//Leak Station Not Homed Timeout
GVL_MASTER.stAlarms[2].aEventTimers[0](IN:= (GVL_Master.stStationSruct[2].nState>=200 AND GVL_Master.stStationSruct[2].nState<=900) ,PT:=T#5S);																	
IF GVL_MASTER.stAlarms[2].aEventTimers[0].Q THEN //
	GVL_MASTER.stAlarms[2].aEventFlags[0] := TRUE;
END_IF
//Leak Station Cycle Timeout
GVL_MASTER.stAlarms[2].aEventTimers[1](IN:= (GVL_Master.stStationSruct[2].nState>1000 AND GVL_Master.stStationSruct[2].nState<2000) ,PT:=T#15S);
IF GVL_MASTER.stAlarms[2].aEventTimers[1].Q THEN // 
	GVL_MASTER.stAlarms[2].aEventFlags[1] := TRUE;
END_IF
//Leak Error
GVL_MASTER.stAlarms[2].aEventTimers[2](IN := (NOT PRG_LeakTest.bLeakTesterNoError),PT:=T#100MS);
IF GVL_MASTER.stAlarms[2].aEventTimers[2].Q THEN //
	GVL_MASTER.stAlarms[2].aEventFlags[2] := TRUE;
END_IF
//Consecutive part rejects
IF PRG_LeakTest.nConsParts>2 THEN // 
	GVL_MASTER.stAlarms[2].aEventFlags[3] := TRUE;
END_IF
END_ACTION

METHOD SetEventTexts : BOOL
VAR_INPUT
END_VAR
//Immediate Faults
GVL_MASTER.stAlarms[2].aEventTexts[0] := 'Leak Station Not Homed Timeout';
GVL_MASTER.stAlarms[2].aEventTexts[1] := 'Leak Station Cycle Timeout';
GVL_MASTER.stAlarms[2].aEventTexts[2] := 'Leak Error';
GVL_MASTER.stAlarms[2].aEventTexts[3] := 'More than 2 Consecutive rejects';
GVL_MASTER.stAlarms[2].aEventTexts[4] := '';
GVL_MASTER.stAlarms[2].aEventTexts[5] := '';
GVL_MASTER.stAlarms[2].aEventTexts[6] := '';
GVL_MASTER.stAlarms[2].aEventTexts[7] := '';
GVL_MASTER.stAlarms[2].aEventTexts[8] := '';
GVL_MASTER.stAlarms[2].aEventTexts[9] := ''; 
GVL_MASTER.stAlarms[2].aEventTexts[10] := ''; 
GVL_MASTER.stAlarms[2].aEventTexts[11] := '';
GVL_MASTER.stAlarms[2].aEventTexts[12] := '';
GVL_MASTER.stAlarms[2].aEventTexts[13] := '';
GVL_MASTER.stAlarms[2].aEventTexts[14] := '';
GVL_MASTER.stAlarms[2].aEventTexts[15] := '';
GVL_MASTER.stAlarms[2].aEventTexts[16] := '';
GVL_MASTER.stAlarms[2].aEventTexts[17] := '';
GVL_MASTER.stAlarms[2].aEventTexts[18] := '';
GVL_MASTER.stAlarms[2].aEventTexts[19] := '';
GVL_MASTER.stAlarms[2].aEventTexts[20] := '';
GVL_MASTER.stAlarms[2].aEventTexts[21] := '';
GVL_MASTER.stAlarms[2].aEventTexts[22] := '';
GVL_MASTER.stAlarms[2].aEventTexts[28] := '';
GVL_MASTER.stAlarms[2].aEventTexts[29] := '';
GVL_MASTER.stAlarms[2].aEventTexts[30] := '';

//Cycle Stop Requests

GVL_MASTER.stAlarms[2].aEventTexts[80] := '';
GVL_MASTER.stAlarms[2].aEventTexts[81] := '';
GVL_MASTER.stAlarms[2].aEventTexts[82] := '';

GVL_MASTER.stAlarms[2].aEventTexts[84] := '';
GVL_MASTER.stAlarms[2].aEventTexts[85] := '';
GVL_MASTER.stAlarms[2].aEventTexts[86] := '';
GVL_MASTER.stAlarms[2].aEventTexts[87] := ''; 
GVL_MASTER.stAlarms[2].aEventTexts[88] := '';
GVL_MASTER.stAlarms[2].aEventTexts[89] := '';

//Master Messages

GVL_MASTER.stAlarms[2].aEventTexts[100] := '';
GVL_MASTER.stAlarms[2].aEventTexts[101] := '';
GVL_MASTER.stAlarms[2].aEventTexts[102] := '';
GVL_MASTER.stAlarms[2].aEventTexts[103] := '';
GVL_MASTER.stAlarms[2].aEventTexts[104] := '';
GVL_MASTER.stAlarms[2].aEventTexts[105] := '';
GVL_MASTER.stAlarms[2].aEventTexts[106] := '';
END_METHOD

END_PROGRAM

// ---- POUs/C_LeakTest/PRG_LeakTest.TcPOU
PROGRAM PRG_LeakTest
VAR
	
		TonCaseDelay  		: ARRAY[1..10] OF Tc2_Standard.TON;
		rtrigCaseTriger  	: ARRAY [1..10] OF Tc2_Standard.R_TRIG;
		
		bLeakTesterNoError	: BOOL;
		uCurrentProgramID	: USINT;
		uSetProgramID		: USINT;
		bProgramAccepted	: BOOL;
		bProgramRejected	: BOOL;
		bInstrumentReady	: BOOL;
		bStart				: BOOL;
		bStop				: BOOL;
		bClearErrorIns		: BOOL;
		bTestActiveLiveData	: BOOL;
		nLiveMeasID			: UDINT;
		nLastMeasID			: UDINT;
		bJobPass			: BOOL;
		bJobFailed			: BOOL;
		nConsParts			: INT;






END_VAR
VAR_IN_OUT
	stStationStruct          : ST_StandardStationStruct;
END_VAR

ACT_IOLink();
ACT_TimTrig();

(************** Station in Home Position **************************)
stStationStruct.bStationHomed :=  (stStationStruct.nState = 1000);

(******************************************************************)
stStationStruct.bStationComplete := stStationStruct.nState = 1900;
stStationStruct.bStationHomingRequest := stStationStruct.nState = 200;
stStationStruct.bStationWaitOnRequest := stStationStruct.nState = 1000; 
stStationStruct.bStationInitDone := stStationStruct.nState = 900;
stStationStruct.bStationInProgressInit := stStationStruct.nState >= 200 AND stStationStruct.nState <= 900;
stStationStruct.bStationInProgress :=  stStationStruct.nState > 1000 AND stStationStruct.nState < 1900;
stStationStruct.bStationWaitOnInit := stStationStruct.nState = 100; 
//stStationStruct.bStationAcknowledge := stStationStruct.nState = 200 OR stStationStruct.nState = 1100;
stStationStruct.bStationNotMoving := stStationStruct.nState = 100 OR stStationStruct.nState = 1000 OR stStationStruct.nState = 1900;
(******************************************************************)
(***************** Counter *************)
IF rtrigCaseTriger[1].Q THEN
GVL_PERSIST.stPartsInspection.nLeakPartsGood:= GVL_PERSIST.stPartsInspection.nLeakPartsGood +1;
GVL_PERSIST.stPartsInspection.nLeakTotalPartsGood := GVL_PERSIST.stPartsInspection.nLeakTotalPartsGood+1;
ELSIF GVL_HMI_GLOBAL.bResetLeakGoodParts THEN
GVL_PERSIST.stPartsInspection.nLeakPartsGood:=0;	
END_IF


IF rtrigCaseTriger[2].Q THEN
	GVL_PERSIST.stPartsInspection.nLeakPartsFailed:=GVL_PERSIST.stPartsInspection.nLeakPartsFailed+1;
	GVL_PERSIST.stPartsInspection.nLeakTotalPartsFailed:= GVL_PERSIST.stPartsInspection.nLeakTotalPartsFailed+1;
ELSIF GVL_HMI_GLOBAL.bResetLeakBadParts THEN
	GVL_PERSIST.stPartsInspection.nLeakPartsFailed:=0;
END_IF


bClearErrorIns := GVL_HMI_GLOBAL.bResetButton;

(***************************************)

IF rtrigCaseTriger[3].Q THEN
	stStationStruct.nState := 100;
END_IF

(***************************************)


CASE stStationStruct.nState OF
100: 
bStart							:= FALSE;
IF stStationStruct.bStationInitRequest THEN
	 stStationStruct.nState := 120;
END_IF
120:
bClearErrorIns := TRUE;
IF bClearErrorIns THEN
	stStationStruct.nState := 160;
END_IF
160:
IF tonCaseDelay[2].Q THEN
	bClearErrorIns := FALSE;
	stStationStruct.nState := 180;
END_IF
180: // Check if error 
IF bLeakTesterNoError THEN
	 stStationStruct.nState := 400;
END_IF
400:
IF tonCaseDelay[1].Q THEN
	stStationStruct.nState := 800;
END_IF
800:
IF bInstrumentReady THEN
	stStationStruct.nState := 900;
END_IF
900:
IF stStationStruct.bStationAcknowledge THEN
	stStationStruct.nState := 1000;
END_IF

1000: // Waiting for request 
IF GVL_HMI_GLOBAL.bResetPassAndFail THEN
	GVL_MASTER.stNest.bLeakPass 	:= FALSE;
   GVL_MASTER.stNest.sLeakHMI 	:= "";
   GVL_MASTER.stNest.bLeakReject := FALSE;
END_IF

IF stStationStruct.bStationRequest AND stStationStruct.bNoCycleStopRequest THEN
   stStationStruct.nState := 1100;  
ELSIF (stStationStruct.bStationManualRequestHMI OR GVL_MASTER.bManualModeTrigger) AND stStationStruct.bNoCycleStopRequest THEN
   stStationStruct.nState := 4000; // Manual Mode
ELSIF stStationStruct.bStationAbort THEN
	   stStationStruct.nState := 100;	   
END_IF
1100: // Check Ready
bStart						:= FALSE;
GVL_MASTER.stNest.bLeakPass := FALSE;
GVL_MASTER.stNest.sLeakHMI 	:= "";
IF bInstrumentReady THEN
	stStationStruct.nState := 1140; 
ELSE
	stStationStruct.nState := 100;
END_IF
1140://Check status of intrument
IF bLeakTesterNoError THEN
	stStationStruct.nState := 1200;
END_IF
1200: 
bStart := TRUE;
IF  tonCaseDelay[3].Q THEN
	stStationStruct.nState := 1220;
END_IF
1220:
bStart := FALSE;
IF  NOT bTestActiveLiveData THEN
	stStationStruct.nState := 1280;
END_IF


1280: // JOB PASS / JOB FAIL
IF bJobPass  THEN
	GVL_MASTER.stNest.bLeakPass := TRUE;
	GVL_MASTER.stNest.sLeakHMI 	:= "Pass";
	GVL_MASTER.stNest.bLeakReject := FALSE;
   	stStationStruct.nState := 1900;
ELSIF bJobFailed  THEN
   stStationStruct.nState := 1900;
   GVL_MASTER.stNest.bLeakPass := FALSE;
   GVL_MASTER.stNest.sLeakHMI 	:= "Fail";
   GVL_MASTER.stNest.bLeakReject := TRUE;
END_IF

1900:
IF (tonCaseDelay[4].Q AND NOT stStationStruct.bStationManualRequestHMI) OR stStationStruct.bNoCycleStopRequest THEN
	stStationStruct.nState := 1000;
ELSIF tonCaseDelay[4].Q AND stStationStruct.bStationManualRequestHMI THEN
	stStationStruct.nState := 4000;
ELSIF stStationStruct.bStationAbort AND tonCaseDelay[2].Q THEN
	stStationStruct.nState := 100;

END_IF
//=== Manual Mode ===
4000:
IF NOT stStationStruct.bStationManualRequestHMI AND NOT GVL_MASTER.bManualModeTrigger THEN
	stStationStruct.nState := 1000;
ELSIF stStationStruct.bStationAbort THEN
	   stStationStruct.nState := 100;	
END_IF
IF GVL_HMI_GLOBAL.bStartLeakMan THEN
	
	bStart 						:= TRUE;
ELSIF GVL_HMI_GLOBAL.bStopLeakMan THEN
	
	bStop						:= TRUE;

ELSE 
	bStart						:= FALSE;
	bStop						:= FALSE;
END_IF
ACT_ChangeJOB();

9000:

bClearErrorIns 					:= FALSE;
bStart							:= FALSE;
GVL_MASTER.stNest.bLeakPass 	:= FALSE;


stStationStruct.nState := 9100;	
9100:
IF tonCaseDelay[5].Q THEN
	stStationStruct.nState := 9200;
END_IF
9200:
bClearErrorIns := TRUE;
IF tonCaseDelay[6].Q THEN
	stStationStruct.nState := 9300;
END_IF
9300: 
IF bLeakTesterNoError THEN
   stStationStruct.nState := 1000;
END_IF

	
END_CASE

IF NOT bLeakTesterNoError AND NOT stStationStruct.nState >= 9000 THEN
stStationStruct.nState := 9000;
END_IF

ACTION ACT_ChangeJob:
	
GVL_IO.dw_B07_i28General_I_O.bSetProgram[0] := GVL_HMI_GLOBAL.uNewLeakProgID.0;
GVL_IO.dw_B07_i28General_I_O.bSetProgram[1] := GVL_HMI_GLOBAL.uNewLeakProgID.1;
GVL_IO.dw_B07_i28General_I_O.bSetProgram[2] := GVL_HMI_GLOBAL.uNewLeakProgID.2;
GVL_IO.dw_B07_i28General_I_O.bSetProgram[3] := GVL_HMI_GLOBAL.uNewLeakProgID.3;
GVL_IO.dw_B07_i28General_I_O.bSetProgram[4] := GVL_HMI_GLOBAL.uNewLeakProgID.4;
GVL_IO.dw_B07_i28General_I_O.bSetProgram[5] := GVL_HMI_GLOBAL.uNewLeakProgID.5;
GVL_IO.dw_B07_i28General_I_O.bSetProgram[6] := GVL_HMI_GLOBAL.uNewLeakProgID.6;
GVL_IO.dw_B07_i28General_I_O.bSetProgram[7] := GVL_HMI_GLOBAL.uNewLeakProgID.7;


IF GVL_HMI_GLOBAL.bSetLeakProgramID THEN 
	
		uSetProgramID := GVL_HMI_GLOBAL.uNewLeakProgID;
END_IF
END_ACTION

ACTION ACT_IOLINK:


bLeakTesterNoError				:= NOT GVL_IO.dw_B07_i28General_I_O.bMalfunction;
uCurrentProgramID				:= GVL_IO.dw_B07_i28General_I_O.nCurrentProgramNumber;
bProgramAccepted				:= GVL_IO.dw_B07_i28General_I_O.bProgramAccept;
bInstrumentReady				:= GVL_IO.dw_B07_i28General_I_O.bInstrumentReady;
bProgramRejected				:= GVL_IO.dw_B07_i28General_I_O.bProgramReject;
bTestActiveLiveData				:= GVL_IO.dw_B07_i28General_I_O.bTestActiveLiveData;
nLiveMeasID						:= GVL_IO.dw_B07_i28LiveMeasurement.inUniqueID;
nLastMeasID						:= GVL_IO.dw_B07_i28LastResult.inUniqueID;
bJobPass						:= GVL_IO.dw_B07_i28General_I_O.bProgramAccept;
bJobFailed						:= GVL_IO.dw_B07_i28General_I_O.bProgramReject;



GVL_IO.dw_B07_i28General_I_O.bStart 			:= bStart;
GVL_IO.dw_B07_i28General_I_O.bStop				:= bStop;
GVL_IO.dw_B07_i28General_I_O.bChangeProgram := GVL_HMI_GLOBAL.bSetLeakProgramID;
GVL_IO.dw_B07_i28General_I_O.bReset := bClearErrorIns OR GVL_HMI_GLOBAL.bResetLeakMan;
END_ACTION

ACTION ACT_TimTrig:


tonCaseDelay[1](IN:= (stStationStruct.nState=400),PT:=T#50MS);
tonCaseDelay[2](IN:= (stStationStruct.nState=160),PT:=T#50MS);
tonCaseDelay[3](IN:= (stStationStruct.nState=1200),PT:=T#10S);
tonCaseDelay[4](IN:= (stStationStruct.nState=1900),PT:=T#1S);
tonCaseDelay[5](IN:= (stStationStruct.nState=9100),PT:=T#200MS);
tonCaseDelay[6](IN:= (stStationStruct.nState=9200),PT:=T#250MS);
tonCaseDelay[7](IN:= ,PT:=T#500MS);



rtrigCaseTriger[1](clk:= (stStationStruct.nState=1900) AND bJobPass);
rtrigCaseTriger[2](clk:= (stStationStruct.nState=1900) AND bJobFailed);
rtrigCaseTriger[3](clk:= stStationStruct.bStationAbort);
END_ACTION

END_PROGRAM

// ---- POUs/D_VisionTest/PRG_Fault_VisionTest.TcPOU
PROGRAM PRG_Fault_VisionTest
VAR
	
			i				: INT;
			
END_VAR
VAR_IN_OUT

  aAlarms  : ARRAY[0..3] OF ST_Events;
END_VAR

ACT_FaultTrig();

(************************************** Faults reset **********************************************)
IF   GVL_HMI_GLOBAL.bResetButton THEN 
	FOR i := 0 TO 127 DO
		GVL_MASTER.stAlarms[3].aEventFlags[i] := FALSE;
	END_FOR
END_IF
//===============================================================
//Initialize event texts on first scan
IF NOT GVL_MASTER.stAlarms[3].bEventTextsSet THEN
	SetEventTexts();
	GVL_MASTER.stAlarms[3].bEventTextsSet := TRUE;
END_IF


(***************************************************************************************************)
//Immediate fault
GVL_MASTER.stAlarms[3].bImmediateFault := FALSE;
FOR i := 0 TO 32DO
	GVL_MASTER.stAlarms[3].bImmediateFault := GVL_MASTER.stAlarms[3].bImmediateFault OR GVL_MASTER.stAlarms[3].aEventFlags[i];
END_FOR

//Cycle stop fault
GVL_MASTER.stAlarms[3].bCycleStopFault := FALSE;
FOR i := 33 TO 79 DO
	GVL_MASTER.stAlarms[3].bCycleStopFault := GVL_MASTER.stAlarms[3].bCycleStopFault OR GVL_MASTER.stAlarms[3].aEventFlags[i];
END_FOR
//Cycle stop Request
GVL_MASTER.stAlarms[3].bCycleStopRequest := FALSE;
FOR i := 80 TO 99 DO
	GVL_MASTER.stAlarms[3].bCycleStopRequest := GVL_MASTER.stAlarms[3].bCycleStopRequest OR GVL_MASTER.stAlarms[3].aEventFlags[i];
END_FOR

ACTION ACT_FaultTrig:
(**************************************************************************************************)
(**************************** Master Immediate Fault Stop *****************************************)
(**************************************************************************************************)
(* Copy Safety Immediate Stop Faults to Master Immediate Stop Faults *)
(* *)

//Camera Station Not Homed Timeout
GVL_MASTER.stAlarms[3].aEventTimers[0](IN:= (GVL_Master.stStationSruct[3].nState>=200 AND GVL_Master.stStationSruct[3].nState<=900) ,PT:=T#5S);																	
IF GVL_MASTER.stAlarms[3].aEventTimers[0].Q THEN //
	GVL_MASTER.stAlarms[3].aEventFlags[0] := TRUE;
END_IF
//Camera Station Cycle Timeout
GVL_MASTER.stAlarms[3].aEventTimers[1](IN:= (GVL_Master.stStationSruct[3].nState>=1100 AND GVL_Master.stStationSruct[3].nState<1900) ,PT:=T#5S);
IF GVL_MASTER.stAlarms[3].aEventTimers[1].Q THEN // 
	GVL_MASTER.stAlarms[3].aEventFlags[1] := TRUE;
END_IF
//Camera Error
GVL_MASTER.stAlarms[3].aEventTimers[2](IN := (NOT PRG_VisionTest.bCamerraNoError),PT:=T#100MS);
IF GVL_MASTER.stAlarms[3].aEventTimers[2].Q THEN //
	GVL_MASTER.stAlarms[3].aEventFlags[2] := TRUE;
END_IF
//Consecutive part rejects
(*IF PRG_VisionTest.nConsParts>2 THEN // 
	GVL_MASTER.stAlarms[3].aEventFlags[3] := TRUE;
END_IF*)

//Adquisition error
IF GVL_IO.dw_B06_IS2802M.aqsAcquisitionError  THEN
	GVL_MASTER.stAlarms[3].aEventFlags[100] := TRUE;
ELSIF NOT GVL_IO.dw_B06_IS2802M.aqsAcquisitionError THEN
   	GVL_MASTER.stAlarms[3].aEventFlags[100] := FALSE;
END_IF
END_ACTION

METHOD PRIVATE SetEventTexts : BOOL
VAR_INPUT
END_VAR
//Immediate Faults
GVL_MASTER.stAlarms[3].aEventTexts[0] := 'Camera Station Not Homed Timeout';
GVL_MASTER.stAlarms[3].aEventTexts[1] := 'Camera Station Cycle Timeout';
GVL_MASTER.stAlarms[3].aEventTexts[2] := 'Camera Error';
//GVL_MASTER.stAlarms[3].aEventTexts[3] := 'More than 2 Consecutive rejects';
GVL_MASTER.stAlarms[3].aEventTexts[4] := '';
GVL_MASTER.stAlarms[3].aEventTexts[5] := '';
GVL_MASTER.stAlarms[3].aEventTexts[6] := '';
GVL_MASTER.stAlarms[3].aEventTexts[7] := '';
GVL_MASTER.stAlarms[3].aEventTexts[8] := '';
GVL_MASTER.stAlarms[3].aEventTexts[9] := ''; 
GVL_MASTER.stAlarms[3].aEventTexts[10] := ''; 
GVL_MASTER.stAlarms[3].aEventTexts[11] := '';
GVL_MASTER.stAlarms[3].aEventTexts[12] := '';
GVL_MASTER.stAlarms[3].aEventTexts[13] := '';
GVL_MASTER.stAlarms[3].aEventTexts[14] := '';
GVL_MASTER.stAlarms[3].aEventTexts[15] := '';
GVL_MASTER.stAlarms[3].aEventTexts[16] := '';
GVL_MASTER.stAlarms[3].aEventTexts[17] := '';
GVL_MASTER.stAlarms[3].aEventTexts[18] := '';
GVL_MASTER.stAlarms[3].aEventTexts[19] := '';
GVL_MASTER.stAlarms[3].aEventTexts[20] := '';
GVL_MASTER.stAlarms[3].aEventTexts[21] := '';
GVL_MASTER.stAlarms[3].aEventTexts[22] := '';
GVL_MASTER.stAlarms[3].aEventTexts[28] := '';
GVL_MASTER.stAlarms[3].aEventTexts[29] := '';
GVL_MASTER.stAlarms[3].aEventTexts[30] := '';

//Cycle Stop Requests

GVL_MASTER.stAlarms[3].aEventTexts[80] := '';
GVL_MASTER.stAlarms[3].aEventTexts[81] := '';
GVL_MASTER.stAlarms[3].aEventTexts[82] := '';

GVL_MASTER.stAlarms[3].aEventTexts[84] := '';
GVL_MASTER.stAlarms[3].aEventTexts[85] := '';
GVL_MASTER.stAlarms[3].aEventTexts[86] := '';
GVL_MASTER.stAlarms[3].aEventTexts[87] := ''; 
GVL_MASTER.stAlarms[3].aEventTexts[88] := '';
GVL_MASTER.stAlarms[3].aEventTexts[89] := '';

//Master Messages

GVL_MASTER.stAlarms[3].aEventTexts[100] := 'Acquisition Error';
GVL_MASTER.stAlarms[3].aEventTexts[101] := '';
GVL_MASTER.stAlarms[3].aEventTexts[102] := '';
GVL_MASTER.stAlarms[3].aEventTexts[103] := '';
GVL_MASTER.stAlarms[3].aEventTexts[104] := '';
GVL_MASTER.stAlarms[3].aEventTexts[105] := '';
GVL_MASTER.stAlarms[3].aEventTexts[106] := '';
END_METHOD

END_PROGRAM

// ---- POUs/D_VisionTest/PRG_VisionTest.TcPOU
PROGRAM PRG_VisionTest
VAR

	biClamp				: BOOL;

	rTrigJobChangeReq	: R_TRIG;
	rTrigProdJob		: R_TRIG;
	rTrigCalibJob		: R_TRIG;

	bCommandExecuting	: BOOL;
	bCommandFailed		: BOOL;
	bCommandCompleted 	: BOOL;
	bCommandExecute		: BOOL;
	nCommandID			: UINT;
	bCamerraNoError     : BOOL;
	bCameraBufOverR     : BOOL;
	bInspectionCompleted: RS;
	bResultValid        : BOOL;
	bJobPass            : BOOL;
	bAqusError          : BOOL;
	bExposComplete      : BOOL;
	bAqusTriggerReady   : BOOL;
	bOnline             : BOOL;
	bOffline            : BOOL;
	bEnableTrigger      : BOOL;
	bTriggerCam         : BOOL;
	bComplete           : BOOL;
	bClearCamError      : BOOL;
	bAcnwResult         : BOOL;
	nCammeraErrorID     : UINT;	
	nAqusID             : UINT;
	nCurrentJobID       : UINT;	
	nRempAqusID         : UINT;
	nCameraJob          : UINT := 1;
	nAqusID_Temp        : UINT := 0;
	bManPass            : BOOL;
	bManFail            : BOOL;
	bManEnablTrig       : BOOL;
	bManTrigCam         : BOOL;
	bManAknwResult      : BOOL;
	bManComplResl       : BOOL;	
	
	nCoutAqErr			: INT;

		
	TonCaseDelay  		: ARRAY[1..10] OF Tc2_Standard.TON;
	rtrigCaseTriger  	: ARRAY [1..10] OF Tc2_Standard.R_TRIG;
	adbCaseFlag      	: ARRAY [1..10] OF BOOL;
	eCamJobState		: E_CameraJobChange;

	nConsParts			: INT;
END_VAR

VAR_IN_OUT
	stStationStruct     : ST_StandardStationStruct;
END_VAR

ACT_IOLink();
ACT_ChangeJob();
ACT_TimTrig();

(************** Station in Home Position **************************)
stStationStruct.bStationHomed :=  (stStationStruct.nState = 1000);

(******************************************************************)
stStationStruct.bStationComplete := stStationStruct.nState = 1900;
stStationStruct.bStationHomingRequest := stStationStruct.nState = 200;
stStationStruct.bStationWaitOnRequest := stStationStruct.nState = 1000; 
stStationStruct.bStationInitDone := stStationStruct.nState = 900;
stStationStruct.bStationInProgressInit := stStationStruct.nState >= 200 AND stStationStruct.nState <= 900;
stStationStruct.bStationInProgress :=  stStationStruct.nState > 1000 AND stStationStruct.nState < 1900;
stStationStruct.bStationWaitOnInit := stStationStruct.nState = 100; 
//stStationStruct.bStationAcknowledge := stStationStruct.nState = 200 OR stStationStruct.nState = 1100;
stStationStruct.bStationNotMoving := stStationStruct.nState = 100 OR stStationStruct.nState = 1000 OR stStationStruct.nState = 1900;
(******************************************************************)
(***************** Counter *************)
IF rtrigCaseTriger[3].Q THEN
GVL_PERSIST.stPartsInspection.nVisionPartsGood:= GVL_PERSIST.stPartsInspection.nVisionPartsGood +1;
GVL_PERSIST.stPartsInspection.nVisionTotalPartsGood := GVL_PERSIST.stPartsInspection.nVisionTotalPartsGood+1;
ELSIF GVL_HMI_GLOBAL.bResetVisionGoodParts THEN
GVL_PERSIST.stPartsInspection.nVisionPartsGood:=0;	
END_IF


IF rtrigCaseTriger[4].Q THEN
	GVL_PERSIST.stPartsInspection.nVisionPartsFailed:=GVL_PERSIST.stPartsInspection.nVisionPartsFailed+1;
	GVL_PERSIST.stPartsInspection.nVisionTotalPartsFailed:= GVL_PERSIST.stPartsInspection.nVisionTotalPartsFailed+1;
ELSIF GVL_HMI_GLOBAL.bResetVisionBadParts THEN
	GVL_PERSIST.stPartsInspection.nVisionPartsFailed:=0;
END_IF

IF rtrigCaseTriger[4].Q THEN
	nConsParts:= nConsParts+1;
ELSIF rtrigCaseTriger[3].Q OR GVL_HMI_GLOBAL.bResetButton THEN
    nConsParts:=0;	
END_IF

bClearCamError := GVL_HMI_GLOBAL.bResetButton;

(***************************************)

IF rtrigCaseTriger[5].Q THEN
	stStationStruct.nState := 100;
END_IF

(***************************************)


CASE stStationStruct.nState OF
100: 
IF stStationStruct.bStationInitRequest THEN
	 stStationStruct.nState := 140;
END_IF
140:
bClearCamError := TRUE;
IF bClearCamError THEN
	stStationStruct.nState := 160;
END_IF
160:
IF tonCaseDelay[8].Q THEN
	bClearCamError := FALSE;
	stStationStruct.nState := 200;
END_IF
200: // Check if error 
IF bCamerraNoError THEN
	 stStationStruct.nState := 400;
END_IF
300: // Check ID job
IF nCurrentJobID = nCameraJob THEN
	stStationStruct.nState := 400;
END_IF
400:
IF tonCaseDelay[1].Q THEN
	stStationStruct.nState := 900;
END_IF
900:
IF stStationStruct.bStationAcknowledge THEN
	stStationStruct.nState := 1000;
END_IF
1000: // Waiting for request 
adbCaseFlag[1] := FALSE;
adbCaseFlag[2] := FALSE;
bEnableTrigger := FALSE;
bTriggerCam    := FALSE;

bAcnwResult := FALSE;
bComplete:= FALSE;
IF GVL_HMI_GLOBAL.bResetPassAndFail THEN
	GVL_MASTER.stNest.bVisionPass := FALSE;
	GVL_MASTER.stNest.sVisionHMI := "";
	GVL_MASTER.stNest.bVisionReject := FALSE;
END_IF
IF stStationStruct.bStationRequest AND stStationStruct.bNoCycleStopRequest THEN
   stStationStruct.nState := 1100;  
ELSIF (stStationStruct.bStationManualRequestHMI OR GVL_MASTER.bManualModeTrigger) AND stStationStruct.bNoCycleStopRequest THEN
   stStationStruct.nState := 4000; // Manual Mode
ELSIF stStationStruct.bStationAbort THEN
	   stStationStruct.nState := 100;	   
END_IF
1100:// Check Buffer
IF NOT bCameraBufOverR THEN
	stStationStruct.nState := 1160;
ELSIF bCameraBufOverR THEN
	stStationStruct.nState := 1120;  
END_IF
1120: 
bOffline := TRUE;
IF NOT bOnline THEN
	bClearCamError := TRUE;
	stStationStruct.nState := 1130; 
END_IF
1130:
IF bClearCamError THEN
	bClearCamError := FALSE;
	stStationStruct.nState := 1140;
END_IF
1140:
IF NOT bClearCamError THEN
       bOffline := FALSE;
       stStationStruct.nState := 1160; 
END_IF
1160: // Check ofline/online
IF bOnline THEN
	stStationStruct.nState := 1200; 
ELSE
	adbCaseFlag[1] := TRUE;
    stStationStruct.nState := 1200; 
END_IF
1180://Check status if Cam
IF nCammeraErrorID =0 THEN
	stStationStruct.nState := 1200;
ELSE
    adbCaseFlag[2] := TRUE;	
	stStationStruct.nState := 2000;
END_IF
1200://Enable Trigger
bEnableTrigger := TRUE;
IF bAqusTriggerReady THEN
	stStationStruct.nState := 1220;
END_IF
1220: 
bTriggerCam := TRUE;
IF  bExposComplete THEN
	stStationStruct.nState := 1240;
END_IF
1240:
IF bResultValid THEN
	bEnableTrigger := FALSE;
	bTriggerCam := FALSE;
	stStationStruct.nState := 1260;
END_IF
1260:// Check Aqusition
IF nAqusID<> nAqusID_Temp AND bInspectionCompleted.Q1 THEN
	stStationStruct.nState := 1270;
END_IF
1270:
IF tonCaseDelay[9].Q THEN
	stStationStruct.nState := 1280;
END_IF

1280: // JOB PASS / JOB FAIL
IF bJobPass  THEN
//   nPartStatus := 1;
	GVL_MASTER.stNest.bVisionPass 	:= TRUE;
	GVL_MASTER.stNest.sVisionHMI 	:= "Pass";
   stStationStruct.nState := 1300;
ELSIF NOT bJobPass  THEN
	//Added checks here not initial for bNestFail or bNestPartReject	
//   nPartStatus := 0;
   GVL_MASTER.stNest.bVisionReject := TRUE;
   GVL_MASTER.stNest.sVisionHMI 	:= "Fail";
   stStationStruct.nState := 1282;
END_IF
1282:
bAcnwResult := TRUE;
IF NOT bResultValid THEN
	stStationStruct.nState := 1284;
END_IF
1284:
bAcnwResult := FALSE;
IF NOT bAcnwResult AND NOT bResultValid THEN
	nAqusID_Temp:= nAqusID;
	stStationStruct.nState := 1286;
END_IF
1286:
bComplete:= TRUE;
IF NOT bExposComplete THEN
	stStationStruct.nState := 1288;
END_IF
1288:
bComplete:= FALSE;
IF NOT bComplete AND NOT bExposComplete THEN
	stStationStruct.nState := 1290;
END_IF	
1290:
adbCaseFlag[1] := FALSE;
adbCaseFlag[2] := FALSE;
bEnableTrigger := FALSE;
bTriggerCam    := FALSE;
bAcnwResult := FALSE;
bComplete:= FALSE;
stStationStruct.nState := 1292;
1292:
bEnableTrigger := TRUE;
IF bEnableTrigger AND tonCaseDelay[7].Q THEN
	stStationStruct.nState := 1294;
END_IF
1294:
bTriggerCam := TRUE;
IF  bExposComplete THEN
	stStationStruct.nState := 1296;
END_IF
1296:
IF bResultValid THEN
	bEnableTrigger := FALSE;
    bTriggerCam := FALSE;
    stStationStruct.nState := 1298;
END_IF
1298:
IF bJobPass  THEN
//   nPartStatus := 1;
   stStationStruct.nState := 1300;
ELSIF NOT  bJobPass THEN
//   nPartStatus := 0;
   stStationStruct.nState := 1300;
END_IF

1300:
bAcnwResult := TRUE;
IF NOT bResultValid THEN
	stStationStruct.nState := 1320;
END_IF
1320:
bAcnwResult := FALSE;
IF NOT bAcnwResult AND NOT bResultValid THEN
	nAqusID_Temp:= nAqusID;
	stStationStruct.nState := 1340;
END_IF
1340:
bComplete:= TRUE;
IF NOT bExposComplete THEN
	stStationStruct.nState := 1360;
END_IF
1360:
bComplete:= FALSE;
IF NOT bComplete AND NOT bExposComplete THEN
	stStationStruct.nState := 1900;
END_IF	
1900:
adbCaseFlag[1] := FALSE;
adbCaseFlag[2] := FALSE;
bEnableTrigger := FALSE;
bTriggerCam    := FALSE;
bAcnwResult := FALSE;
bComplete:= FALSE;
IF tonCaseDelay[2].Q AND rtrigCaseTriger[7].Q THEN
	stStationStruct.nState := 1000;
ELSIF NOT stStationStruct.bNoCycleStopRequest AND tonCaseDelay[2].Q THEN
	stStationStruct.nState := 1000;
END_IF
//=== Manual Mode ===
4000:
IF NOT stStationStruct.bStationManualRequestHMI  AND NOT GVL_MASTER.bManualModeTrigger THEN
	stStationStruct.nState := 1000;
END_IF
IF GVL_HMI_GLOBAL.bEnableTrigerMan THEN
	bManEnablTrig := TRUE;
	bManPass:= FALSE;
	bManFail:= FALSE;
	stStationStruct.nState := 4100;
ELSIF stStationStruct.bStationAbort THEN
	   stStationStruct.nState := 100;		
END_IF
4100:
	bManPass:= FALSE;
	bManFail:= FALSE;
IF NOT stStationStruct.bStationManualRequestHMI THEN
	bManEnablTrig := FALSE;
	stStationStruct.nState := 1000;
ELSIF stStationStruct.bStationAbort THEN
	   bManEnablTrig := FALSE;
	   stStationStruct.nState := 100;		
ELSIF GVL_HMI_GLOBAL.bTrigerCamMan THEN
	GVL_HMI_GLOBAL.bEnableTrigerMan:= FALSE;
	bManTrigCam := TRUE;
	stStationStruct.nState := 4200;
END_IF
4200:
GVL_HMI_GLOBAL.bTrigerCamMan := FALSE;
IF  bExposComplete THEN
	stStationStruct.nState := 4300;
END_IF
4300:
IF bResultValid THEN
	bManEnablTrig := FALSE;
    bManTrigCam := FALSE;
    stStationStruct.nState := 4400;
END_IF
4400:
IF bJobPass THEN
	bManPass := TRUE;
	bManFail := FALSE;
//	nPartStatus := 1;
	stStationStruct.nState := 4500;
ELSIF NOT bJobPass  THEN
	bManPass := FALSE;
	bManFail := TRUE;
//	nPartStatus := 0;
	stStationStruct.nState := 4500;
END_IF
4500:
bManAknwResult := TRUE;
IF NOT bResultValid THEN
	stStationStruct.nState := 4600;
END_IF
4600:
bManAknwResult := FALSE;
bManComplResl := TRUE;
IF NOT bExposComplete THEN
	stStationStruct.nState := 4700;
END_IF
4700:
bManAknwResult := FALSE;
bManComplResl  := FALSE;
bManEnablTrig  := FALSE;
bManTrigCam    := FALSE;
IF NOT stStationStruct.bStationManualRequestHMI THEN
stStationStruct.nState := 4000;
ELSE
stStationStruct.nState := 1000;	
END_IF
9000:

bManAknwResult := FALSE;
bManComplResl  := FALSE;
bManEnablTrig  := FALSE;
bManTrigCam    := FALSE;	
bOffline       := FALSE;
bEnableTrigger := FALSE;
bTriggerCam    := FALSE;
bComplete      := FALSE;
bClearCamError := FALSE;
bAcnwResult    := FALSE;
stStationStruct.nState := 9100;	
9100:
IF tonCaseDelay[5].Q THEN
	stStationStruct.nState := 9200;
END_IF
9200:
bClearCamError := TRUE;
IF tonCaseDelay[6].Q THEN
	stStationStruct.nState := 9300;
END_IF
9300: 
IF nCoutAqErr >3 THEN
   stStationStruct.nState := 1000;
ELSIF nCoutAqErr <=3 THEN
   stStationStruct.nState := 1100;
END_IF

	
END_CASE

IF bAqusError AND NOT stStationStruct.nState >= 9000 THEN
stStationStruct.nState := 9000;
END_IF


IF rtrigCaseTriger[6].Q THEN
   nCoutAqErr := nCoutAqErr +1;
ELSIF  stStationStruct.nState = 1000 THEN
    nCoutAqErr := 0;
END_IF

ACTION ACT_ChangeJob:
rTrigProdJob(CLK := GVL_HMI_GLOBAL.bLoadProductionJob);
rTrigCalibJob(CLK := GVL_HMI_GLOBAL.bLoadCalibrationJob);

IF rTrigProdJob.Q THEN
	eCamJobState := E_CameraJobChange.LOAD_PROD_JOB;
END_IF

IF rTrigCalibJob.Q THEN
	eCamJobState := E_CameraJobChange.LOAD_CALB_JOB;
END_IF

CASE eCamJobState OF
	
E_CameraJobChange.WAITING_FOR_REQUEST:
//Do nothing

E_CameraJobChange.LOAD_PROD_JOB:
	(*Load Production Job*)
	nCommandID := 1;
	eCamJobState := E_CameraJobChange.GO_OFFLINE;

E_CameraJobChange.LOAD_CALB_JOB:
	(*Load Calibration Job*)
	nCommandID := 101;
	eCamJobState := E_CameraJobChange.GO_OFFLINE;

E_CameraJobChange.GO_OFFLINE:
	bOffline := TRUE;
	eCamJobState := E_CameraJobChange.EXECUTE_COMMAND;

E_CameraJobChange.EXECUTE_COMMAND:
	bCommandExecute := TRUE;
	eCamJobState := E_CameraJobChange.RESET_FLAG;
	
E_CameraJobChange.RESET_FLAG:
IF bCommandCompleted THEN
	bCommandExecute := FALSE;
	bOffline := FALSE;
	GVL_HMI_GLOBAL.bLoadProductionJob := FALSE;
	GVL_HMI_GLOBAL.bLoadCalibrationJob := FALSE;
	eCamJobState := E_CameraJobChange.WAITING_FOR_REQUEST;
END_IF
END_CASE
END_ACTION

ACTION ACT_IOLink:

bCamerraNoError      := NOT GVL_IO.dw_B06_IS2802M.isError;//==
nCammeraErrorID      := GVL_IO.dw_B06_IS2802M.isErrorID;//--nchamera UI
bCameraBufOverR      := GVL_IO.dw_B06_IS2802M.isResultsBufferOverrun;
bInspectionCompleted(SET := GVL_IO.dw_B06_IS2802M.isInspectionCompleted, RESET1 := stStationStruct.nState > 1260);
bResultValid         := GVL_IO.dw_B06_IS2802M.isResultsValid;
bJobPass             := GVL_IO.dw_B06_IS2802M.isJobPassed;
bAqusError           := GVL_IO.dw_B06_IS2802M.aqsAcquisitionError;
bExposComplete       := GVL_IO.dw_B06_IS2802M.aqsExposureComplete;
bAqusTriggerReady    := GVL_IO.dw_B06_IS2802M.aqsTriggerReady;
bOnline              := GVL_IO.dw_B06_IS2802M.aqsOnline;
nAqusID              := GVL_IO.dw_B06_IS2802M.aqsAcquisitionID;
nCurrentJobID        := GVL_IO.dw_B06_IS2802M.ccoCurrentJobID;
bCommandExecuting	 := GVL_IO.dw_B06_IS2802M.isCommandExecuting;
bCommandFailed		 := GVL_IO.dw_B06_IS2802M.isCommandFailed;
bCommandCompleted    := GVL_IO.dw_B06_IS2802M.isCommandCompleted;
GVL_IO.dw_B06_IS2802M.aqcSetOffline                  := bOffline;
GVL_IO.dw_B06_IS2802M.aqcTriggerEnable               := bEnableTrigger OR bManEnablTrig;
GVL_IO.dw_B06_IS2802M.aqcTrigger                     := bTriggerCam OR bManTrigCam;
GVL_IO.dw_B06_IS2802M.aqcClearExposureComplete       := bComplete OR bManComplResl;
GVL_IO.dw_B06_IS2802M.icClearError                   := bClearCamError OR GVL_HMI_GLOBAL.bResetCamMan ;//--
GVL_IO.dw_B06_IS2802M.icInspectionResultsAcknowledge := bAcnwResult OR bManAknwResult ;
GVL_IO.dw_B06_IS2802M.cciCommandID					 := nCommandID;
GVL_IO.dw_B06_IS2802M.icExecuteCommand				 := bCommandExecute;

biClamp					:= GVL_IO.dw_T02_EL1809.iCalmpClosed;

IF tonCaseDelay[4].Q THEN
	GVL_HMI_GLOBAL.bResetCamMan:= FALSE;
END_IF

IF NOT bExposComplete THEN
   bComplete:= FALSE;
END_IF
IF bExposComplete THEN
	bTriggerCam := FALSE;
END_IF
IF NOT bResultValid THEN
	bAcnwResult := FALSE;
END_IF

IF NOT GVL_Master.stMachineStatus.bManualMode THEN
   GVL_HMI_GLOBAL.sInfoCamMan:= 'Machine not in Manual Mode';
ELSIF GVL_Master.stMachineStatus.bManualMode AND stStationStruct.nState>4100 THEN
   GVL_HMI_GLOBAL.sInfoCamMan:= 'Camera in Process';
ELSIF  GVL_Master.stMachineStatus.bManualMode AND stStationStruct.nState=4000 THEN
   GVL_HMI_GLOBAL.sInfoCamMan:= 'Waiting for Enable'; 
ELSIF  GVL_Master.stMachineStatus.bManualMode AND stStationStruct.nState=4100 THEN
   GVL_HMI_GLOBAL.sInfoCamMan:= 'Waiting for Trigger';		   
END_IF
END_ACTION

ACTION ACT_TimTrig:
tonCaseDelay[1](IN:= (stStationStruct.nState=400),PT:=T#50MS);
tonCaseDelay[2](IN:= (stStationStruct.nState=1900),PT:=T#100MS);
tonCaseDelay[3](IN:= (stStationStruct.nState=1),PT:=T#100MS);
tonCaseDelay[4](IN:= GVL_HMI_GLOBAL.bResetCamMan,PT:=T#100MS);
tonCaseDelay[5](IN:= (stStationStruct.nState=9100),PT:=T#250MS);
tonCaseDelay[6](IN:= (stStationStruct.nState=9200),PT:=T#250MS);
tonCaseDelay[7](IN:= (stStationStruct.nState=1292),PT:=T#50MS);
tonCaseDelay[8](IN:= (stStationStruct.nState=160),PT:=T#250MS);
tonCaseDelay[9](IN:=stStationStruct.nState=1270 ,PT:=T#1S);
tonCaseDelay[10](IN:= ,PT:=T#250MS);

rtrigCaseTriger[1](clk:= stStationStruct.nState>1100);
rtrigCaseTriger[2](clk:= adbCaseFlag[1]);
rtrigCaseTriger[3](clk:= (stStationStruct.nState=1900) AND bJobPass );
rtrigCaseTriger[4](clk:= (stStationStruct.nState=1900) AND NOT bJobPass );
rtrigCaseTriger[5](clk:= stStationStruct.bStationAbort);
rtrigCaseTriger[6](clk:= (stStationStruct.nState=1240) AND  bAqusError );
rtrigCaseTriger[7](clk:= biClamp);
rtrigCaseTriger[8](clk:= );
rtrigCaseTriger[9](clk:= );
rtrigCaseTriger[10](clk:= );
END_ACTION

END_PROGRAM

// ---- POUs/A_Master/PRG_MachineStatus.TcPOU
PROGRAM PRG_MachineStatus
VAR

	tonPowerUp						: TON;
	tonSystemInitialising			: TON;
	tonSystemInitialisingTimeout	: TON;
	
	bMemoSystemReadyToStart			:BOOL; //flag set only once to establissh if system was in ready to start state after powerUP
	
// =========== Manual =============	

	rtrigManualModeOFF              :ARRAY[1..4] OF R_TRIG;
	rtrigManualMode                 :R_TRIG;	
		// =========== Master Time =============
		//Variables
	bReadyToRead				:BOOL;
	bFirstScan					:BOOL := TRUE;
	bUpdateSysTime				:BOOL; //Output of pulse generator
	tSysTimeUpdatePeriod		:TIME := T#5S;
	stTimeStamp					:TIMESTRUCT;
	stNullTimeStamp				:TIMESTRUCT;
	sRawDateTime				:STRING;

	

	
	
	sDateTime					:STRING;
	sDateTimeSpaces				:STRING;
	
	
	
	//Functions
	fbGetSystemTime				:TC2_Utilities.NT_GetTime;
	fbRTClock					:TC2_Utilities.RTC_EX2;		//Local real-time clock
	tonTimeUpdateGen			:TC2_Utilities.TON;			//Pulse generator for triggering fbGetSystemTime function
	rtrigSysTimeCollected		:TC2_Utilities.R_TRIG;		//System time collected



		
END_VAR

ACT_ManualMode();
ACT_MasterTime();
ACT_MachineStatusBaner();


(*Power Up*)

tonPowerUp( IN := TRUE,  PT := T#5S, Q => GVL_MASTER.stMasterControl.bPowerUpTimerComplete );

(*System Initialising*)

tonSystemInitialising( IN := (GVL_MASTER.stMachineStatus.eMachineState = E_MachineState.SYSTEM_INITIALISING),
	PT := T#1S,
	Q => GVL_MASTER.stMasterControl.bSystemInitialisingTimerComplete);
	
(*System Initialising Timeout*)
	
tonSystemInitialisingTimeout(IN := (GVL_MASTER.stMachineStatus.eMachineState = E_MachineState.SYSTEM_INITIALISING),
	PT := T#5M,
	Q => GVL_MASTER.stMasterControl.bSystemInitialisingTimeoutComplete);
	
(* Set Machine State to Power Up while waiting for Power Up Timer to Complete *)
IF NOT GVL_MASTER.stMasterControl.bPowerUpTimerComplete THEN
	GVL_MASTER.stMachineStatus.eMachineState := E_MachineState.SYSTEM_POWER_UP;
END_IF

(********************************(Sequence )*******************************************************)
(* Move to Immediate Stopped once there is an Immediate Fault *)
IF NOT GVL_MASTER.stMasterControl.bNoMachineImmediateFault THEN		
	GVL_MASTER.stMachineStatus.eMachineState := E_MachineState.IMMEDIATE_STOPPED;
ELSIF NOT GVL_MASTER.stMasterControl.bNoCycleStopFault THEN
	GVL_MASTER.stMachineStatus.eMachineState := E_MachineState.CYCLE_STOP_FAULT;	
END_IF

CASE GVL_MASTER.stMachineStatus.eMachineState OF
	
E_MachineState.SYSTEM_POWER_UP:
	
	bMemoSystemReadyToStart:=FALSE;
	(* Move to Immediate Stopped once Power Up Timer has completed *)
	IF GVL_MASTER.stMasterControl.bPowerUpTimerComplete THEN			
		GVL_MASTER.stMachineStatus.eMachineState := E_MachineState.IMMEDIATE_STOPPED;
	END_IF
	
E_MachineState.IMMEDIATE_STOPPED:	
	(* Move to System Initialising once there is no Immediate Fault *)
	IF GVL_MASTER.stMasterControl.bNoMachineImmediateFault  THEN	
		GVL_MASTER.stMachineStatus.eMachineState := E_MachineState.SYSTEM_INITIALISING;
	(* Move to Immediate Fault once there is an Immediate Fault *)
	ELSIF NOT GVL_MASTER.stMasterControl.bNoMachineImmediateFault THEN
		GVL_MASTER.stMachineStatus.eMachineState := E_MachineState.IMMEDIATE_FAULT;	
	END_IF
	
E_MachineState.SYSTEM_INITIALISING:		
	IF  GVL_MASTER.stMasterControl.bNoMachineImmediateFault	 AND GVL_MASTER.stMasterControl.bSystemInitialisingTimerComplete  THEN		
		GVL_MASTER.stMachineStatus.eMachineState := E_MachineState.SYSTEM_READY_TO_START;
	
	//Move to Cycle Stopped once there is a Cycle Stop Request AND All Stations are Cycle Stopped AND there is No Immediate Fault*)
	ELSIF GVL_HMI_GLOBAL.bStopButton
		OR (GVL_MASTER.stMasterControl.bNoMachineImmediateFault 
		AND (GVL_MASTER.stMasterControl.bSystemInitialisingTimeoutComplete OR GVL_MASTER.stMasterControl.bCycleStopRequest) AND GVL_MASTER.stMasterControl.bAllStationsCycledStopped)
	THEN		
		GVL_MASTER.stMachineStatus.eMachineState := E_MachineState.CYCLE_STOPPED;			
	ELSIF GVL_MASTER.stMasterControl.bNoMachineImmediateFault AND NOT GVL_MASTER.stMasterControl.bNoCycleStopFault THEN		
		GVL_MASTER.stMachineStatus.eMachineState := E_MachineState.CYCLE_STOP_FAULT;	
	ELSIF NOT GVL_MASTER.stMasterControl.bNoStationImmediateFault THEN
         GVL_MASTER.stMachineStatus.eMachineState := E_MachineState.IMMEDIATE_FAULT;
      	
	END_IF
	
E_MachineState.SYSTEM_READY_TO_START:
	bMemoSystemReadyToStart := TRUE;
	
	//Move to System Auto if the Start Button has been pressed
	IF GVL_MASTER.stMasterControl.bManualModeRequest THEN
		GVL_MASTER.stMachineStatus.eMachineState := E_MachineState.MANUAL_MODE;
	
	ELSIF GVL_HMI_GLOBAL.bStopButton THEN
        GVL_MASTER.stMachineStatus.eMachineState := E_MachineState.STOPPING; 
	ELSIF GVL_HMI_GLOBAL.bStartButton AND NOT PRG_Mastercycle.biClamp AND NOT PRG_Mastercycle.biPartPresent   THEN			
		GVL_MASTER.stMachineStatus.eMachineState := E_MachineState.SYSTEM_AUTO_CYCLE;
		
	//Move to Cycle Stopped once there is a Cycle Stop Request AND All Stations are Cycle Stopped AND there is No Immediate Fault
	ELSIF (GVL_MASTER.stMasterControl.bCycleStopRequest OR NOT	GVL_MASTER.stMasterControl.bNoCycleStopFault) 
	AND GVL_MASTER.stMasterControl.bNoMachineImmediateFault
	THEN				
		GVL_MASTER.stMachineStatus.eMachineState := E_MachineState.CYCLE_STOPPED;	
	ELSIF NOT GVL_MASTER.stMasterControl.bNoCycleStopFault THEN
		GVL_MASTER.stMachineStatus.eMachineState := E_MachineState.CYCLE_STOP_FAULT;
	ELSIF NOT GVL_MASTER.stMasterControl.bNoMachineImmediateFault OR NOT GVL_MASTER.stMasterControl.bNoStationImmediateFault THEN
       GVL_MASTER.stMachineStatus.eMachineState := E_MachineState.IMMEDIATE_FAULT ;	
	   
	END_IF
	

	
	
	
E_MachineState.SYSTEM_AUTO_CYCLE:	
	//Move to System Dwell once there is a Dwell Request
	IF GVL_MASTER.stMasterControl.bDwellRequest THEN
		GVL_MASTER.stMachineStatus.eMachineState := E_MachineState.SYSTEM_DWELL;
	
	//Move to Cycle Stopped once there is a Cycle Stop Request AND All Stations are Cycle Stopped AND there is No Immediate Fault OR when cycle done
	ELSIF NOT GVL_MASTER.stMasterControl.bNoCycleStopFault THEN //Fast cycle stop	
		GVL_MASTER.stMachineStatus.eMachineState := E_MachineState.CYCLE_STOP_FAULT;
	(*ELSIF GVL_Master.bMachineCycleDone   THEN 
	stMachineStatus.eMachineState := E_MachineState.CYCLE_STOPPED; //Instant cycle stop???		*)
	ELSIF GVL_HMI_GLOBAL.bStopButton OR GVL_MASTER.stMasterControl.bCycleStopRequest OR GVL_HMI_GLOBAL.nRegionMain <> 1 THEN
		GVL_MASTER.stMachineStatus.eMachineState := E_MachineState.STOPPING; //Stopping sequence 
	ELSIF NOT GVL_MASTER.stMasterControl.bNoStationImmediateFault OR NOT GVL_MASTER.stMasterControl.bNoMachineImmediateFault THEN
		GVL_MASTER.stMachineStatus.eMachineState := E_MachineState.IMMEDIATE_FAULT;
	END_IF	

E_MachineState.SYSTEM_DWELL:		
	(* Move to System Auto Cycle once the Start Button is Pressed AND there is No Dwell Request *)
	IF NOT GVL_MASTER.stMasterControl.bDwellRequest THEN
		GVL_MASTER.stMachineStatus.eMachineState := E_MachineState.SYSTEM_AUTO_CYCLE;	
	(* Move to Cycle Stopped once there is a Cycle Stop Request AND All Stations are Cycle Stopped AND there is No Immediate Fault*)
	ELSIF (GVL_MASTER.stMasterControl.bCycleStopRequest OR	NOT	GVL_MASTER.stMasterControl.bNoCycleStopFault) 
		AND GVL_MASTER.stMasterControl.bAllStationsCycledStopped AND GVL_MASTER.stMasterControl.bNoMachineImmediateFault
	THEN				
		GVL_MASTER.stMachineStatus.eMachineState := E_MachineState.CYCLE_STOPPED;	
	END_IF

E_MachineState.STOPPING: 
	IF  GVL_MASTER.stMasterControl.bAllStationsCycledStopped THEN
		GVL_MASTER.stMachineStatus.eMachineState := E_MachineState.CYCLE_STOPPED;
	ELSIF NOT GVL_MASTER.stMasterControl.bNoCycleStopFault THEN
		GVL_MASTER.stMachineStatus.eMachineState := E_MachineState.CYCLE_STOP_FAULT;
	ELSIF NOT GVL_MASTER.stMasterControl.bNoMachineImmediateFault OR NOT GVL_MASTER.stMasterControl.bNoStationImmediateFault THEN
        GVL_MASTER.stMachineStatus.eMachineState := E_MachineState.IMMEDIATE_FAULT ;
	END_IF
	
E_MachineState.CYCLE_STOPPED:
	IF GVL_MASTER.stMasterControl.bManualModeRequest THEN
		GVL_MASTER.stMachineStatus.eMachineState := E_MachineState.MANUAL_MODE;			
	(* Move to System Initialising once there is no Cycle Stop Fault AND the Reset Button is Pressed *)
	ELSIF (GVL_MASTER.stMasterControl.bNoCycleStopFault AND GVL_HMI_GLOBAL.bResetButton )THEN
		GVL_MASTER.stMachineStatus.eMachineState := E_MachineState.SYSTEM_INITIALISING;		
	ELSIF NOT GVL_MASTER.stMasterControl.bNoStationImmediateFault THEN
       	GVL_MASTER.stMachineStatus.eMachineState := E_MachineState.IMMEDIATE_FAULT;
	END_IF	

E_MachineState.CYCLE_STOP_FAULT:	
	(* Move to Cycle Stopped once there no Cycle Stop Fault AND there is No Immediate Fault*)
	IF GVL_MASTER.stMasterControl.bNoCycleStopFault THEN
		GVL_MASTER.stMachineStatus.eMachineState := E_MachineState.CYCLE_STOPPED;
	END_IF	
ELSE 	
	GVL_MASTER.stMachineStatus.eMachineState := E_MachineState.SYSTEM_POWER_UP;	
	
E_MachineState.MANUAL_MODE:

	IF NOT GVL_MASTER.stMasterControl.bManualModeRequest THEN
		GVL_MASTER.stMachineStatus.eMachineState := E_MachineState.CYCLE_STOPPED;
	END_IF
	
E_MachineState.IMMEDIATE_FAULT:		
	(* Move to Immediate Stopped once there is an Immediate Fault *)
	IF GVL_MASTER.stMasterControl.bNoMachineImmediateFault AND  GVL_MASTER.stMasterControl.bNoStationImmediateFault THEN
		GVL_MASTER.stMachineStatus.eMachineState := E_MachineState.IMMEDIATE_STOPPED;		

	END_IF
END_CASE
//////////////////////////////////////////////////////////////////////////////////////////////////////////////
								//CYCLE STOP REQUEST//
//////////////////////////////////////////////////////////////////////////////////////////////////////////////
IF GVL_MASTER.stAlarms[0].bCycleStopRequest OR GVL_MASTER.stAlarms[1].bCycleStopRequest OR GVL_MASTER.stAlarms[2].bCycleStopRequest OR GVL_MASTER.stAlarms[3].bCycleStopRequest THEN
				GVL_MASTER.stMasterControl.bCycleStopRequest	:=	TRUE;
ELSE			GVL_MASTER.stMasterControl.bCycleStopRequest	:=	FALSE;
END_IF




(************************************* write all system states to variables ***********************)

GVL_MASTER.stMachineStatus.bSystemPowerUp :=(GVL_MASTER.stMachineStatus.eMachineState = E_MachineState.SYSTEM_POWER_UP);
GVL_MASTER.stMachineStatus.bImmediateStopped :=(GVL_MASTER.stMachineStatus.eMachineState = E_MachineState.IMMEDIATE_STOPPED);
GVL_MASTER.stMachineStatus.bSystemInitialising :=(GVL_MASTER.stMachineStatus.eMachineState = E_MachineState.SYSTEM_INITIALISING);
GVL_MASTER.stMachineStatus.bSystemReadyToStart := (GVL_MASTER.stMachineStatus.eMachineState = E_MachineState.SYSTEM_READY_TO_START);
GVL_MASTER.stMachineStatus.bSystemAutoCycle := (GVL_MASTER.stMachineStatus.eMachineState = E_MachineState.SYSTEM_AUTO_CYCLE);
GVL_MASTER.stMachineStatus.bSystemDwell := (GVL_MASTER.stMachineStatus.eMachineState = E_MachineState.SYSTEM_DWELL);
GVL_MASTER.stMachineStatus.bSystemStopping := (GVL_MASTER.stMachineStatus.eMachineState = E_MachineState.STOPPING);
GVL_MASTER.stMachineStatus.bCycleStopped := (GVL_MASTER.stMachineStatus.eMachineState = E_MachineState.CYCLE_STOPPED);
GVL_MASTER.stMachineStatus.bManualMode := (GVL_MASTER.stMachineStatus.eMachineState = E_MachineState.MANUAL_MODE);
GVL_MASTER.stMachineStatus.bImmediateFault := (GVL_MASTER.stMachineStatus.eMachineState = E_MachineState.IMMEDIATE_FAULT);
GVL_MASTER.stMachineStatus.bCycleStopFault := (GVL_MASTER.stMachineStatus.eMachineState = E_MachineState.CYCLE_STOP_FAULT);

ACTION ACT_MachineStatusBaner:
//Machine status banner action
//SYSTEM POWER UP
IF GVL_MASTER.stMachineStatus.bSystemPowerUp THEN	
	GVL_MASTER.stMachineStatus.sMachineStatusText := 'SYSTEM POWER UP';		// fill colour WHITE, text colour BLACK
	GVL_MASTER.stMachineStatus.nMachineStatusColour := nWHITE;
	GVL_MASTER.stMachineStatus.nMachineStatusTxtCol := nBLACK;
	GVL_MASTER.stMachineStatus.sBannerBckColor := sWHITE;
	GVL_MASTER.stMachineStatus.sBannerTextColor := sBLACK;
END_IF

(* IMMEDIATE STOPPED *)
IF GVL_MASTER.stMachineStatus.bImmediateStopped THEN	
	GVL_MASTER.stMachineStatus.sMachineStatusText := 'IMMEDIATE STOPPED';		// fill colour BLACK, text colour WHITE
	GVL_MASTER.stMachineStatus.nMachineStatusColour := nBLACK;
	GVL_MASTER.stMachineStatus.nMachineStatusTxtCol := nWHITE;
	GVL_MASTER.stMachineStatus.sBannerBckColor := sBLACK;
	GVL_MASTER.stMachineStatus.sBannerTextColor := sWHITE;	
END_IF

(* SYSTEM INITIALISING *)
IF GVL_MASTER.stMachineStatus.bSystemInitialising THEN	
	GVL_MASTER.stMachineStatus.sMachineStatusText := 'SYSTEM INITIALIZING';		// fill colour YELLOW, text colour BLACK
	GVL_MASTER.stMachineStatus.nMachineStatusColour := nYELLOW;
	GVL_MASTER.stMachineStatus.nMachineStatusTxtCol := nBLACK;
	GVL_MASTER.stMachineStatus.sBannerBckColor := sYELLOW;
	GVL_MASTER.stMachineStatus.sBannerTextColor := sBLACK;
END_IF
(*
(* SYSTEM IN STANDBY *)
IF stMachineStatus.bSystemStandby THEN
	stMachineStatus.sMachineStatusText := 'SYSTEM IN STANDBY';
	stMachineStatus.nMachineStatusColour := nORANGE;
	stMachineStatus.nMachineStatusTxtCol := nWHITE;
END_IF
*)
(* SYSTEM READY TO START FLASH ON *)
IF GVL_MASTER.stMachineStatus.bSystemReadyToStart AND GVL_MASTER.bFlash1Hz THEN
	GVL_MASTER.stMachineStatus.sMachineStatusText := 'SYSTEM READY TO START';		// fill colour GREEN, text colour WHITE
	GVL_MASTER.stMachineStatus.nMachineStatusColour := nGREEN;
	GVL_MASTER.stMachineStatus.nMachineStatusTxtCol := nWHITE;
	GVL_MASTER.stMachineStatus.sBannerBckColor := sGREEN;
	GVL_MASTER.stMachineStatus.sBannerTextColor := sWHITE;
END_IF

(* SYSTEM READY TO START FLASH OFF *)
IF GVL_MASTER.stMachineStatus.bSystemReadyToStart AND NOT GVL_MASTER.bFlash1Hz THEN	
	GVL_MASTER.stMachineStatus.sMachineStatusText := 'SYSTEM READY TO START';		// fill colour WHITE, text colour GREEN
	GVL_MASTER.stMachineStatus.nMachineStatusColour := nWHITE;
	GVL_MASTER.stMachineStatus.nMachineStatusTxtCol := nGREEN;
	GVL_MASTER.stMachineStatus.sBannerBckColor := sWHITE;
	GVL_MASTER.stMachineStatus.sBannerTextColor := sGREEN;
END_IF

(* SYSTEM AUTO CYCLE *)
IF GVL_MASTER.stMachineStatus.bSystemAutoCycle THEN	
	GVL_MASTER.stMachineStatus.sMachineStatusText := 'SYSTEM AUTO CYCLE';		// fill colour GREEN, text colour WHITE
	GVL_MASTER.stMachineStatus.nMachineStatusColour := nGREEN;
	GVL_MASTER.stMachineStatus.nMachineStatusTxtCol := nWHITE;
	GVL_MASTER.stMachineStatus.sBannerBckColor := sGREEN;
	GVL_MASTER.stMachineStatus.sBannerTextColor := sWHITE;	
END_IF

(* SYSTEM DWELL *)
IF GVL_MASTER.stMachineStatus.bSystemDwell THEN	
	GVL_MASTER.stMachineStatus.sMachineStatusText := 'SYSTEM DWELL';		// fill colour ORANGE, text colourWHITE
	GVL_MASTER.stMachineStatus.nMachineStatusColour := nORANGE;
	GVL_MASTER.stMachineStatus.nMachineStatusTxtCol := nWHITE;
	GVL_MASTER.stMachineStatus.sBannerBckColor := sORANGE;
	GVL_MASTER.stMachineStatus.sBannerTextColor := sWHITE;	
END_IF

(* STOPPING *)
IF GVL_MASTER.stMachineStatus.bSystemStopping AND GVL_MASTER.bFlash1Hz THEN	
	GVL_MASTER.stMachineStatus.sMachineStatusText := 'STOPPING';		// fill colour BLACK, text colour WHITE
	GVL_MASTER.stMachineStatus.nMachineStatusColour := nBLACK;
	GVL_MASTER.stMachineStatus.nMachineStatusTxtCol := nWHITE;
	GVL_MASTER.stMachineStatus.sBannerBckColor := sBLACK;
	GVL_MASTER.stMachineStatus.sBannerTextColor := sWHITE;	
END_IF

(* STOPPING *)
IF GVL_MASTER.stMachineStatus.bSystemStopping AND NOT GVL_MASTER.bFlash1Hz THEN	
	GVL_MASTER.stMachineStatus.sMachineStatusText := 'STOPPING';		// fill colour WHITE, text colour BLACK
	GVL_MASTER.stMachineStatus.nMachineStatusColour := nWHITE;
	GVL_MASTER.stMachineStatus.nMachineStatusTxtCol := nBLACK;
	GVL_MASTER.stMachineStatus.sBannerBckColor := sWHITE;
	GVL_MASTER.stMachineStatus.sBannerTextColor := sBLACK;	
END_IF

(* CYCLE STOPPED *)
IF GVL_MASTER.stMachineStatus.bCycleStopped THEN	
	GVL_MASTER.stMachineStatus.sMachineStatusText := 'CYCLE STOPPED';		// fill colour BLACK, text colour WHITE
	GVL_MASTER.stMachineStatus.nMachineStatusColour := nBLACK;
	GVL_MASTER.stMachineStatus.nMachineStatusTxtCol := nWHITE;
	GVL_MASTER.stMachineStatus.sBannerBckColor := sBLACK;
	GVL_MASTER.stMachineStatus.sBannerTextColor := sWHITE;	
END_IF

(* IMMEDIATE FAULT FLASH ON *)
IF GVL_MASTER.stMachineStatus.bImmediateFault AND GVL_MASTER.bFlash1Hz THEN	
	GVL_MASTER.stMachineStatus.sMachineStatusText := 'IMMEDIATE FAULT';		// fill colour RED, text colour WHITE
	GVL_MASTER.stMachineStatus.nMachineStatusColour := nRED;
	GVL_MASTER.stMachineStatus.nMachineStatusTxtCol := nWHITE;
	GVL_MASTER.stMachineStatus.sBannerBckColor := sRED;
	GVL_MASTER.stMachineStatus.sBannerTextColor := sWHITE;	
END_IF

(* IMMEDIATE FAULT FLASH OFF *)
IF GVL_MASTER.stMachineStatus.bImmediateFault AND NOT GVL_MASTER.bFlash1Hz THEN	
	GVL_MASTER.stMachineStatus.sMachineStatusText := 'IMMEDIATE FAULT';		// fill colour WHITE, text colour BLACK
	GVL_MASTER.stMachineStatus.nMachineStatusColour := nWHITE;
	GVL_MASTER.stMachineStatus.nMachineStatusTxtCol := nBLACK;
	GVL_MASTER.stMachineStatus.sBannerBckColor := sWHITE;
	GVL_MASTER.stMachineStatus.sBannerTextColor := sBLACK;	
END_IF

(* CYCLE STOP FAULT FLASH ON *)
IF GVL_MASTER.stMachineStatus.bCycleStopFault AND GVL_MASTER.bFlash1Hz THEN	
	GVL_MASTER.stMachineStatus.sMachineStatusText := 'CYCLE STOP FAULT';		// fill colour RED, text colour WHITE
	GVL_MASTER.stMachineStatus.nMachineStatusColour := nRED;
	GVL_MASTER.stMachineStatus.nMachineStatusTxtCol := nWHITE;
	GVL_MASTER.stMachineStatus.sBannerBckColor := sRED;
	GVL_MASTER.stMachineStatus.sBannerTextColor := sWHITE;	
END_IF

(* CYCLE STOP FAULT FLASH OFF *)
IF GVL_MASTER.stMachineStatus.bCycleStopFault AND NOT GVL_MASTER.bFlash1Hz THEN	
	GVL_MASTER.stMachineStatus.sMachineStatusText := 'CYCLE STOP FAULT';		// fill colour WHITE, text colour RED
	GVL_MASTER.stMachineStatus.nMachineStatusColour := nWHITE;
	GVL_MASTER.stMachineStatus.nMachineStatusTxtCol := nRED;
	GVL_MASTER.stMachineStatus.sBannerBckColor := sWHITE;
	GVL_MASTER.stMachineStatus.sBannerTextColor := sRED;	
END_IF

(* MANUAL MODE *)
IF GVL_MASTER.stMachineStatus.bManualMode THEN	
	GVL_MASTER.stMachineStatus.sMachineStatusText := 'MANUAL MODE';		// fill colour BLUE text colour WHITE
	GVL_MASTER.stMachineStatus.nMachineStatusColour := nBLUE;
	GVL_MASTER.stMachineStatus.nMachineStatusTxtCol := nWHITE;
	GVL_MASTER.stMachineStatus.sBannerBckColor := sBLUE;
	GVL_MASTER.stMachineStatus.sBannerTextColor := sWHITE;	
END_IF

(*
(* SYSTEM READY TO START FLASH ON *)
IF stMachineStatus.bSystemPurge AND bFlash1Hz THEN
	stMachineStatus.sMachineStatusText := 'SYSTEM PURGE';		// fill colour GREEN, text colour WHITE
	stMachineStatus.nMachineStatusColour := nORANGE;
	stMachineStatus.nMachineStatusTxtCol := nBLACK;
	stMachineStatus.sBannerBckColor := sORANGE;
	stMachineStatus.sBannerTextColor := sBLACK;	
END_IF

(* SYSTEM READY TO START FLASH OFF *)
IF stMachineStatus.bSystemPurge AND NOT bFlash1Hz THEN	
	stMachineStatus.sMachineStatusText := 'SYSTEM PURGE';		// fill colour WHITE, text colour GREEN
	stMachineStatus.nMachineStatusColour := nWHITE;
	stMachineStatus.nMachineStatusTxtCol := nBLUE;
	stMachineStatus.sBannerBckColor := sWHITE;
	stMachineStatus.sBannerTextColor := sBLUE;	
END_IF
*)
(*
(* CALIBRATION *)
IF stMachineStatus.bCalibrationFlag AND bFlash1Hz THEN	
	stMachineStatus.sMachineStatusText := 'CALIBRATION MODE';		// fill colour BLUE text colour WHITE
	stMachineStatus.nMachineStatusColour := nBLUE;
	stMachineStatus.nMachineStatusTxtCol := nWHITE;
	stMachineStatus.sBannerBckColor := sBLUE;
	stMachineStatus.sBannerTextColor := sWHITE;	
END_IF
IF stMachineStatus.bCalibrationFlag AND NOT bFlash1Hz THEN	
	stMachineStatus.sMachineStatusText := 'CALIBRATION MODE';		// fill colour BLUE text colour WHITE
	stMachineStatus.nMachineStatusColour := nWHITE;
	stMachineStatus.nMachineStatusTxtCol := nBLUE;
	stMachineStatus.sBannerBckColor := sWHITE;
	stMachineStatus.sBannerTextColor := sBLUE;	
END_IF
*)
END_ACTION

ACTION ACT_ManualMode:
IF	 GVL_MASTER.stMachineStatus.bSystemReadyToStart THEN
	GVL_HMI_GLOBAL.bEnableManualMode := TRUE;
ELSE GVL_HMI_GLOBAL.bEnableManualMode := FALSE;
END_IF


rtrigManualMode(CLK:= GVL_HMI_GLOBAL.nRegionMain=10);
rtrigManualModeOFF[1](CLK:=GVL_Master.stMachineStatus.bManualMode AND (GVL_HMI_GLOBAL.nRegionMain <> 10));
rtrigManualModeOFF[2](CLK:=GVL_Master.stMachineStatus.bManualMode AND GVL_HMI_GLOBAL.bStopButton);
rtrigManualModeOFF[3](CLK:=GVL_Master.stMachineStatus.bManualMode AND NOT GVL_Master.stMasterControl.bNoStationImmediateFault );
rtrigManualModeOff[4](CLK := GVL_HMI_GLOBAL.bManualModeOff[1], Q => GVL_HMI_GLOBAL.bManualModeOff[2]);

IF rtrigManualMode.Q THEN 
	GVL_Master.stMasterControl.bManualModeRequest := TRUE;
	GVL_HMI_GLOBAL.bManualModeOff[1] := FALSE;
ELSIF rtrigManualModeOFF[1].Q OR rtrigManualModeOFF[2].Q OR rtrigManualModeOFF[3].Q THEN
	GVL_Master.stMasterControl.bManualModeRequest := FALSE ;
	GVL_HMI_GLOBAL.bManualModeOff[1] := TRUE;
	
ELSE GVL_HMI_GLOBAL.bManualModeOff[1] := FALSE;
	
END_IF





IF GVL_Master.stMachineStatus.bManualMode  THEN
	GVL_Master.stStationSruct[1].bStationManualRequestHMI := TRUE;
	GVL_Master.stStationSruct[2].bStationManualRequestHMI := TRUE;
	GVL_Master.stStationSruct[3].bStationManualRequestHMI := TRUE;
ELSE
    GVL_Master.stStationSruct[1].bStationManualRequestHMI := FALSE;
	GVL_Master.stStationSruct[2].bStationManualRequestHMI := FALSE;
	GVL_Master.stStationSruct[3].bStationManualRequestHMI := FALSE;	
END_IF
END_ACTION

ACTION ACT_MasterTime:
//Aux functions call
tonTimeUpdateGen(	IN := NOT bUpdateSysTime,
					PT := tSysTimeUpdatePeriod,
					Q => bUpdateSysTime);

//bReadyToRead :=  Tc2_System.MEMCMP( ADR( stTimeStamp), ADR (stNullTimeStamp), SIZEOF(stTimeStamp)) <> 0 AND NOT  fbGetSystemTime.BUSY;	
			(*keczi*)	(*zrobione po to zeby w wypadku jak po starcie PLC na HMI mial pokazywac czas alarmu '00:00:00', zebyb poczekal az faktycznie pokazuje date i czas*)

//Get Current System Time
fbGetSystemTime(NETID := ,
				START := bFirstScan OR bUpdateSysTime,
				TMOUT := ,
				BUSY => ,
				ERR => ,
				ERRID => ,
				TIMESTR => );
				
//Get system time done detection - one-shot
rtrigSysTimeCollected(CLK := NOT fbGetSystemTime.BUSY);

//Synchronize Real-Time clock with system time
fbRTClock(	EN := rtrigSysTimeCollected.Q, 
			PDT := fbGetSystemTime.TIMESTR,
			CDT => stTimeStamp, 
			Q => bReadyToRead);

// System Date and Time in Proper Order 
IF bReadyToRead THEN
	sRawDateTime := SYSTEMTIME_TO_STRING(stTimeStamp);  // format: YYYY-MM-DD-hh:mm:ss.xxx
	GVL_HMI_GLOBAL.sSystemDate := CONCAT(CONCAT(CONCAT(CONCAT(MID(sRawDateTime, 2, 9), '.'),  MID(sRawDateTime, 2, 6)), '.'), LEFT(sRawDateTime, 4));
	GVL_HMI_GLOBAL.sSystemTime := MID(sRawDateTime, 8, 12);
	sDateTime := CONCAT(CONCAT(GVL_HMI_GLOBAL.sSystemDate, '  '), GVL_HMI_GLOBAL.sSystemTime);
	sDateTimeSpaces	:= CONCAT(sDateTime, '    ');
END_IF;

bFirstScan := FALSE;
END_ACTION

END_PROGRAM

// ---- POUs/E_HMI/PRG_HMI.TcPOU
PROGRAM PRG_HMI
VAR
	

	tonCaseDelay				: ARRAY [1..20] OF TON;
	tofCase						: ARRAY [1..20] OF TOF;
	rtrigCaseTriger				: ARRAY [1..20] OF R_TRIG;

	tonResetStatistics			: TON;
END_VAR

ACT_ScreensNamesSet();
ACT_Buttons();
ACT_TimTrig();
ACT_General();

tonResetStatistics( IN := 	GVL_HMI_GLOBAL.aResetHeightSensorBadParts [1] 	OR
							GVL_HMI_GLOBAL.aResetHeightSensorBadParts [2] 	OR
							GVL_HMI_GLOBAL.aResetHeightSensorBadParts [3] 	OR
							GVL_HMI_GLOBAL.aResetHeightSensorBadParts [4] 	OR
							GVL_HMI_GLOBAL.aResetHeightSensorGoodParts[1]	OR
							GVL_HMI_GLOBAL.aResetHeightSensorGoodParts[2]	OR
							GVL_HMI_GLOBAL.aResetHeightSensorGoodParts[3]	OR
							GVL_HMI_GLOBAL.aResetHeightSensorGoodParts[4]	OR
							GVL_HMI_GLOBAL.bResetHeightFailParts			OR
							GVL_HMI_GLOBAL.bResetHeightGoodParts			OR
							GVL_HMI_GLOBAL.bResetGoodParts					OR
							GVL_HMI_GLOBAL.bResetLeakBadParts				OR
							GVL_HMI_GLOBAL.bResetLeakGoodParts				OR
							GVL_HMI_GLOBAL.bResetVisionBadParts				OR
							GVL_HMI_GLOBAL.bResetVisionGoodParts			OR
							GVL_HMI_GLOBAL.bResetFailedParts				OR
							GVL_HMI_GLOBAL.bResetGoodParts					,
							PT												:= T#500MS);

ACTION ACT_Buttons:
ACT_TimTrig();

IF tonCaseDelay[1].Q THEN
	
		GVL_HMI_GLOBAL.bResetButton	:= FALSE;
		
END_IF
IF tonCaseDelay[2].Q THEN
	
		GVL_HMI_GLOBAL.bStopButton	:= FALSE;
		
END_IF
IF tonCaseDelay[3].Q THEN
	
		GVL_HMI_GLOBAL.bStartButton	:= FALSE;
		
END_IF

IF GVL_HMI_GLOBAL.bStartLeakMan THEN
	GVL_IO.dw_B07_i28General_I_O.bStart := TRUE;
END_IF
IF tonCaseDelay[4].Q THEN
	
		GVL_HMI_GLOBAL.bStartLeakMan	:= FALSE;
		GVL_IO.dw_B07_i28General_I_O.bStart := FALSE;
END_IF

IF GVL_HMI_GLOBAL.bStopLeakMan THEN
	GVL_IO.dw_B07_i28General_I_O.bStop := TRUE;
END_IF
IF tonCaseDelay[5].Q THEN
	
		GVL_HMI_GLOBAL.bStopLeakMan	:= FALSE;
		GVL_IO.dw_B07_i28General_I_O.bStop := FALSE;
		
END_IF

IF GVL_HMI_GLOBAL.bResetLeakMan THEN
	GVL_IO.dw_B07_i28General_I_O.bReset := TRUE;
END_IF
IF tonCaseDelay[6].Q THEN
	
		GVL_HMI_GLOBAL.bResetLeakMan	:= FALSE;
		GVL_IO.dw_B07_i28General_I_O.bReset := FALSE;
		
END_IF

IF tonCaseDelay[7].Q THEN
	
		GVL_HMI_GLOBAL.bShutDown	:= FALSE;
		
END_IF
IF tonCaseDelay[8].Q THEN
	
		GVL_HMI_GLOBAL.bSetLeakProgramID	:= FALSE;
		
END_IF

IF tonCaseDelay[9].Q THEN
	
		GVL_HMI_GLOBAL.bSetSetPointsHeightTest	:= FALSE;
		
END_IF

IF tonCaseDelay[10].Q THEN
	
		GVL_HMI_GLOBAL.bManualMeasureHeightTest	:= FALSE;
		
END_IF

IF tonResetStatistics.Q THEN
	
							GVL_HMI_GLOBAL.aResetHeightSensorBadParts [1] 	:= FALSE;
							GVL_HMI_GLOBAL.aResetHeightSensorBadParts [2] 	:= FALSE;
							GVL_HMI_GLOBAL.aResetHeightSensorBadParts [3] 	:= FALSE;
							GVL_HMI_GLOBAL.aResetHeightSensorBadParts [4] 	:= FALSE;
							GVL_HMI_GLOBAL.aResetHeightSensorGoodParts[1]	:= FALSE;
							GVL_HMI_GLOBAL.aResetHeightSensorGoodParts[2]	:= FALSE;
							GVL_HMI_GLOBAL.aResetHeightSensorGoodParts[3]	:= FALSE;
							GVL_HMI_GLOBAL.aResetHeightSensorGoodParts[4]	:= FALSE;
							GVL_HMI_GLOBAL.bResetHeightFailParts			:= FALSE;
							GVL_HMI_GLOBAL.bResetHeightGoodParts			:= FALSE;
							GVL_HMI_GLOBAL.bResetGoodParts					:= FALSE;
							GVL_HMI_GLOBAL.bResetLeakBadParts				:= FALSE;
							GVL_HMI_GLOBAL.bResetLeakGoodParts				:= FALSE;
							GVL_HMI_GLOBAL.bResetVisionBadParts				:= FALSE;
							GVL_HMI_GLOBAL.bResetVisionGoodParts			:= FALSE;
							GVL_HMI_GLOBAL.bResetFailedParts				:= FALSE;
							GVL_HMI_GLOBAL.bResetGoodParts					:= FALSE;


END_IF
END_ACTION

ACTION ACT_General:
IF tofCase[1].Q AND 
( NOT GVL_MASTER.stMasterControl.bNoStationImmediateFault OR NOT GVL_MASTER.stMasterControl.bNoCycleStopFault) THEN
	GVL_HMI_GLOBAL.bAutocycleFaultDialog := TRUE;
END_IF
END_ACTION

ACTION ACT_ScreensNamesSet:
GVL_HMI_GLOBAL.aIOScreen[0] := 'Overview';
GVL_HMI_GLOBAL.aIOScreen[1] := 'HMI - CP2913-0000 | Beckhoff HMI';
GVL_HMI_GLOBAL.aIOScreen[2] := 'PLC - C6015-0010 | Beckhoff PLC | Windows 10 Embedded';
GVL_HMI_GLOBAL.aIOScreen[3] := 'Terminal 1- EK1100 | EtherCAT Coupler';
GVL_HMI_GLOBAL.aIOScreen[4] := 'Terminal 2 - EL6070 | Licence ';
GVL_HMI_GLOBAL.aIOScreen[5] := CONCAT('Terminal 3 - ' , GVL_IO.dw_T02_EL1809.sTerminalName);
GVL_HMI_GLOBAL.aIOScreen[6] := CONCAT('Terminal 4 - ' , GVL_IO.dw_T03_EL2809.sTerminalName);
GVL_HMI_GLOBAL.aIOScreen[7] := 'Terminal 12 - EL6631 |  2-port communication interface';
GVL_HMI_GLOBAL.aIOScreen[8] := 'DL-PN1 | Keyence Communication Unit | ProfiNET';
GVL_HMI_GLOBAL.aIOScreen[9] := 'IS2802  | Cognex Camera| ProfiNET';
GVL_HMI_GLOBAL.aIOScreen[10] := 'I28 | Cincinnati Leak Tester | ProfiNET';

GVL_HMI_GLOBAL.aManualScreen[0] := 'Cognex | Vision Test';
GVL_HMI_GLOBAL.aManualScreen[1] := 'Keyence | Height Test';
GVL_HMI_GLOBAL.aManualScreen[2] := 'Cincinnati | Leak Test';
END_ACTION

ACTION ACT_TimTrig:


tonCaseDelay[1](IN:= GVL_HMI_GLOBAL.bResetButton,PT:=T#500MS);
tonCaseDelay[2](IN:= GVL_HMI_GLOBAL.bStopButton,PT:=T#500MS);
tonCaseDelay[3](IN:= GVL_HMI_GLOBAL.bStartButton,PT:=T#500MS);
tonCaseDelay[4](IN:= GVL_HMI_GLOBAL.bStartLeakMan,PT:=T#500MS);
tonCaseDelay[5](IN:= GVL_HMI_GLOBAL.bStopLeakMan,PT:=T#500MS);
tonCaseDelay[6](IN:= GVL_HMI_GLOBAL.bResetLeakMan,PT:=T#500MS);
//tonCaseDelay[7](IN:= GVL_HMI_GLOBAL.bShutDown,PT:=T#500MS);
tonCaseDelay[8](IN:= GVL_HMI_GLOBAL.bSetLeakProgramID,PT:=T#5S);
tonCaseDelay[9](IN:= GVL_HMI_GLOBAL.bSetSetPointsHeightTest,PT:=T#1S);
tonCaseDelay[10](IN:= GVL_HMI_GLOBAL.bManualMeasureHeightTest,PT:=T#1S);

tofCase[1](IN:= (GVL_Master.stStationSruct[0].nState > 1000 AND GVL_Master.stStationSruct[0].nState < 1900),PT:=T#1S);


rtrigCaseTriger[1](CLK := GVL_MASTER.stNest.bPieceReject);
END_ACTION

END_PROGRAM

// ---- POUs/C_LeakTest/PRG_LeakTestEvents_Info.TcPOU
PROGRAM PRG_LeakTestEvents_Info
VAR
	
	asLeakTesterSegments 				: ARRAY [0..200] OF WSTRING;
	asLeakTesterTestData 				: ARRAY [0..200] OF WSTRING;
	asLeakTesterUnit 	 				: ARRAY [0..200] OF WSTRING;
	asLeakTesterPrecision				: ARRAY [0..10]  OF WSTRING;
	asLeakTesterProgramEvaluation		: ARRAY [0..20]  OF WSTRING;
	asLeakTesterTestEvaluation			: ARRAY [0..150]  OF WSTRING;
	asLeakTesterTestType				: ARRAY [0..25]  OF WSTRING;
	fLeakTesterActive					: F_TRIG;
	bLeakTesterActive					: BOOL;
	Test1								: BOOL;
	
	i									: DINT;

END_VAR

ACT_LiveSegmentCode();
ACT_LeakTesterTestData();
ACT_LeakTesterUnit();
ACT_Precision();
ACT_ProgramEvaluation();
ACT_LeakTesterTestEvaluation();
ACT_TestType();

//Last Result DATA

GVL_IO.dw_B07_i28LastResult.sPartEvaluation 		:= asLeakTesterTestData[GVL_IO.dw_B07_i28LastResult.inTestType];
GVL_IO.dw_B07_i28LastResult.sPrecision				:= asLeakTesterPrecision[GVL_IO.dw_B07_i28LastResult.inPrecisionCode];
GVL_IO.dw_B07_i28LastResult.sTestType				:= asLeakTesterTestType[ GVL_IO.dw_B07_i28LastResult.inPartEvaluation];
GVL_IO.dw_B07_i28LastResult.sUnit1      			:= asLeakTesterUnit[GVL_IO.dw_B07_i28LastResult.inUnitCode1];
GVL_IO.dw_B07_i28LastResult.sUnit2					:= asLeakTesterUnit[GVL_IO.dw_B07_i28LastResult.inUnitCode2];
GVL_IO.dw_B07_i28LastResult.sVariable1				:= asLeakTesterTestData[GVL_IO.dw_B07_i28LastResult.inVariableCode1];
GVL_IO.dw_B07_i28LastResult.sVariable2				:= asLeakTesterTestData[GVL_IO.dw_B07_i28LastResult.inVariableCode2];

//Live DATA


GVL_IO.dw_B07_i28LiveMeasurement.sPrecision1		:= asLeakTesterPrecision[GVL_IO.dw_B07_i28LiveMeasurement.inPrecisionCode1];
GVL_IO.dw_B07_i28LiveMeasurement.sPrecision2		:= asLeakTesterPrecision[GVL_IO.dw_B07_i28LiveMeasurement.inPrecisionCode2];
GVL_IO.dw_B07_i28LiveMeasurement.sPrecision3		:= asLeakTesterPrecision[GVL_IO.dw_B07_i28LiveMeasurement.inPrecisionCode3];
GVL_IO.dw_B07_i28LiveMeasurement.sPrecision4		:= asLeakTesterPrecision[GVL_IO.dw_B07_i28LiveMeasurement.inPrecisionCode4];
GVL_IO.dw_B07_i28LiveMeasurement.sSegmentCode		:= asLeakTesterSegments[GVL_IO.dw_B07_i28LiveMeasurement.inSegmentCode];
GVL_IO.dw_B07_i28LiveMeasurement.sUnit1				:= asLeakTesterUnit[GVL_IO.dw_B07_i28LiveMeasureMENT.inUnitCode1];
GVL_IO.dw_B07_i28LiveMeasurement.sUnit2				:= asLeakTesterUnit[GVL_IO.dw_B07_i28LiveMeasureMENT.inUnitCode2];
GVL_IO.dw_B07_i28LiveMeasurement.sUnit3				:= asLeakTesterUnit[GVL_IO.dw_B07_i28LiveMeasureMENT.inUnitCode3];
GVL_IO.dw_B07_i28LiveMeasurement.sUnit4				:= asLeakTesterUnit[GVL_IO.dw_B07_i28LiveMeasureMENT.inUnitCode4];
GVL_IO.dw_B07_i28LiveMeasurement.sVariable1			:= asLeakTesterTestData[GVL_IO.dw_B07_i28LiveMeasurement.inVariableCode1];
GVL_IO.dw_B07_i28LiveMeasurement.sVariable2			:= asLeakTesterTestData[GVL_IO.dw_B07_i28LiveMeasurement.inVariableCode2];
GVL_IO.dw_B07_i28LiveMeasurement.sVariable3			:= asLeakTesterTestData[GVL_IO.dw_B07_i28LiveMeasurement.inVariableCode3];
GVL_IO.dw_B07_i28LiveMeasurement.sVariable4			:= asLeakTesterTestData[GVL_IO.dw_B07_i28LiveMeasurement.inVariableCode4];


ACT_LastResultSet();

ACTION ACT_LastResultSet:

fLeakTesterActive(CLK := GVL_IO.dw_B07_i28General_I_O.bTestActiveLiveData, Q => bLeakTesterActive);

IF bLeakTesterActive THEN
	
	FOR i :=200 TO 1 BY (-1) DO
		GVL_PERSIST.ast_i28LasResult[i]	:= GVL_PERSIST.ast_i28LasResult[i-1];
	END_FOR
	
	GVL_PERSIST.ast_i28LasResult[0] := GVL_IO.dw_B07_i28LastResult;
	GVL_PERSIST.ast_i28LasResult[0].sTime := GVL_HMI_GLOBAL.sSystemTime;
	GVL_PERSIST.ast_i28LasResult[0].sDate := GVL_HMI_GLOBAL.sSystemDate;

END_IF
END_ACTION

ACTION ACT_LeakTesterTestData:
asLeakTesterTestData[0] := "NO DATA";
asLeakTesterTestData[1] := "Elapsed Timer";
asLeakTesterTestData[2] := "Segment Timer";
asLeakTesterTestData[3] := "Test Execution Time";
asLeakTesterTestData[4] := "Target Pressure";
asLeakTesterTestData[5] := "Test Pressure";
asLeakTesterTestData[6] := "Master Part Profile Test Pressure";
asLeakTesterTestData[7] := "Master Part & Leak Profile Test Pressure";
asLeakTesterTestData[8] := "Leak Standard Calibrated Pressure";
asLeakTesterTestData[9] := "Self Test Pressure";
asLeakTesterTestData[10] := "Measured Pressure";
asLeakTesterTestData[11] := "Instrument Pressure";
asLeakTesterTestData[12] := "Master Gauge Pressure";
asLeakTesterTestData[13] := "Master Part Pressure Loss (Corrected)";
asLeakTesterTestData[14] := "Low Limit Pressure Loss";
asLeakTesterTestData[15] := "High Limit Pressure Loss";
asLeakTesterTestData[16] := "Master Part & Leak Pressure Loss (Corrected)";
asLeakTesterTestData[17] := "Pressure Loss (Corrected)";
asLeakTesterTestData[18] := "Pressure Loss (Actual Read)";
asLeakTesterTestData[19] := "Master Part Flow Offset (Corrected)";
asLeakTesterTestData[20] := "Performance Factor";
asLeakTesterTestData[21] := "Low Limit Rate";
asLeakTesterTestData[22] := "High Limit Rate";
asLeakTesterTestData[23] := "Loss Rate (Corrected)";
asLeakTesterTestData[24] := "Loss Rate (Actual Read)";
asLeakTesterTestData[25] := "Quik Test Pressure";
asLeakTesterTestData[26] := "Quik Test Loss (Corrected)";
asLeakTesterTestData[27] := "Quik Test Flow (Corrected)";
asLeakTesterTestData[28] := "Low Limit Leak Rate";
asLeakTesterTestData[29] := "High Limit Leak Rate";
asLeakTesterTestData[30] := "Predicted Leak Rate";
asLeakTesterTestData[31] := "Leak Rate";
asLeakTesterTestData[32] := "Corrected Leak Standard Calibrated Flow";
asLeakTesterTestData[33] := "Measured Flow";
asLeakTesterTestData[34] := "Environmental Drift Correction Offset";
asLeakTesterTestData[35] := "Transducer Type";
asLeakTesterTestData[36] := "Transducer Typical Residual";
asLeakTesterTestData[37] := "Transducer Zero Low Window";
asLeakTesterTestData[38] := "Transducer Zero High Window";
asLeakTesterTestData[39] := "Regulator Type";
asLeakTesterTestData[40] := "Analog A/D Value";
asLeakTesterTestData[41] := "Peak Pressure";
asLeakTesterTestData[42] := "Analog Input";
asLeakTesterTestData[43] := "Analog Output";
asLeakTesterTestData[44] := "Event Delta Pressure";
asLeakTesterTestData[45] := "Alternate Leak Rate";
asLeakTesterTestData[46] := "DP Master Part Pressure Loss (Corrected)";
asLeakTesterTestData[47] := "DP Master Part & Leak Pressure Loss (Corrected)";
asLeakTesterTestData[48] := "Master Part Quik Pressure Loss (Corrected)";
asLeakTesterTestData[49] := "Master Part Quik Pressure Loss (Actual Read)";
asLeakTesterTestData[50] := "Master Part & Leak Quik Pressure Loss (Corrected)";
asLeakTesterTestData[51] := "Master Part & Leak Quik Pressure Loss (Actual Read)";
asLeakTesterTestData[52] := "Master Part Quik Test Pressure";
asLeakTesterTestData[53] := "Master Part & Leak Quik Test Pressure";
asLeakTesterTestData[54] := "Master Part Quik DP Pressure Loss (Corrected)";
asLeakTesterTestData[55] := "Master Part Quik DP Pressure Loss (Actual Read)";
asLeakTesterTestData[56] := "Master Part & Leak Quik DP Pressure Loss (Actual Read)";
asLeakTesterTestData[57] := "Signal to Noise Ratio";
asLeakTesterTestData[58] := "Effective Number of Bits";
asLeakTesterTestData[59] := "Flicker Free Number of Bits";
asLeakTesterTestData[60] := "High Limit Percent Volume";
asLeakTesterTestData[61] := "Part Percent Volume";
asLeakTesterTestData[62] := "Reference Pressure";
asLeakTesterTestData[63] := "Fill Pressure";
asLeakTesterTestData[64] := "Transducer Cal/Verify - Number of Points";
asLeakTesterTestData[65] := "Transducer - Setpoint Pressure Value";
asLeakTesterTestData[66] := "Transducer - Instrument Pressure Reading";
asLeakTesterTestData[67] := "Transducer - Instrument Flow Reading";
asLeakTesterTestData[68] := "Transducer - Analog Value";
asLeakTesterTestData[69] := "Transducer - Master Reading";
asLeakTesterTestData[70] := "Transducer - Master Value";
asLeakTesterTestData[71] := "Transducer - Atmospheric Pressure";
asLeakTesterTestData[72] := "Transducer - Linearity";
asLeakTesterTestData[73] := "Electronic Regulator Cal - Number of Points";
asLeakTesterTestData[74] := "Electronic Regulator - Instrument Pressure Reading";
asLeakTesterTestData[75] := "Electronic Regulator - Analog Value";
asLeakTesterTestData[76] := "Electronic Regulator - Master Value";
asLeakTesterTestData[77] := "Electronic Regulator Analysis - Number of Points";
asLeakTesterTestData[78] := "Electronic Regulator Analysis - Instrument Pressure Reading";
asLeakTesterTestData[79] := "Electronic Regulator Analysis - Voltage Low Limit";
asLeakTesterTestData[80] := "Electronic Regulator Analysis - Voltage High Limit";
asLeakTesterTestData[81] := "Event Pressure";
asLeakTesterTestData[82] := "Part Flow";
asLeakTesterTestData[83] := "Pre-Pressure";
asLeakTesterTestData[84] := "Tracer Cumulative Leak Rate";
asLeakTesterTestData[85] := "Sniffer Test Location";
asLeakTesterTestData[86] := "Electronic Regulator Cal - Atmospheric Pressure";
asLeakTesterTestData[87] := "REF External Xdcr Pressure";
asLeakTesterTestData[88] := "Differential Pressure Loss (Corrected)";
asLeakTesterTestData[89] := "Differential Pressure Loss (Actual Read)";
asLeakTesterTestData[90] := "Reference Pressure Loss";
asLeakTesterTestData[91] := "Differential Pressure Loss (Actual Read)";
asLeakTesterTestData[92] := "Input State";
asLeakTesterTestData[93] := "Leak Loss";
asLeakTesterTestData[94] := "Batch Quantity";
asLeakTesterTestData[95] := "DP Leak Loss";
asLeakTesterTestData[96] := "Average Quantity";
asLeakTesterTestData[97] := "Charge Pressure";
asLeakTesterTestData[98] := "Standard Pressure";
asLeakTesterTestData[99] := "Instrument Volume";
asLeakTesterTestData[100] := "Part Volume";
asLeakTesterTestData[101] := "Test Measurement Time";
asLeakTesterTestData[102] := "Calculated Leak Rate Offset";
END_ACTION

ACTION ACT_LeakTesterTestEvaluation:
asLeakTesterTestEvaluation[0] := "NO DATA";
asLeakTesterTestEvaluation[1] := "PROGRAM ACCEPT";
asLeakTesterTestEvaluation[2] := "PROGRAM REJECT";
asLeakTesterTestEvaluation[3] := "PART REJECT - LEVEL 1";
asLeakTesterTestEvaluation[4] := "PART REJECT - LEVEL 2";
asLeakTesterTestEvaluation[5] := "PART REJECT - LEVEL 3";
asLeakTesterTestEvaluation[6] := "PROGRAM CALIBRATION PASSED";
asLeakTesterTestEvaluation[7] := "PROGRAM CALIBRATION FAILED";
asLeakTesterTestEvaluation[8] := "MASTER PART COMPLETE";
asLeakTesterTestEvaluation[9] := "SELF-TEST PASSED";
asLeakTesterTestEvaluation[10] := "SELF-TEST FAILED";
asLeakTesterTestEvaluation[11] := "SEQUENCE COMPLETE";
asLeakTesterTestEvaluation[12] := "SEVERE LEAK";
asLeakTesterTestEvaluation[13] := "TEST PRESSURE LOW";
asLeakTesterTestEvaluation[14] := "TEST PRESSURE HIGH";
asLeakTesterTestEvaluation[15] := "BELOW TARGET PRESSURE";
asLeakTesterTestEvaluation[16] := "ABOVE TARGET PRESSURE";
asLeakTesterTestEvaluation[17] := "HELIUM BACKGROUND FAULT";
asLeakTesterTestEvaluation[18] := "PART EVAC FAULT";
asLeakTesterTestEvaluation[19] := "TRANSDUCER ZERO BAD";
asLeakTesterTestEvaluation[20] := "TRANSDUCER OVER-RANGE";
asLeakTesterTestEvaluation[21] := "FLOW TRANSDUCER ZERO BAD";
asLeakTesterTestEvaluation[22] := "FLOW TRANSDUCER OVER-RANGE";
asLeakTesterTestEvaluation[23] := "ERROR: EXCESSIVE FLOW";
asLeakTesterTestEvaluation[24] := "PROGRAM CONFIGURATION ERROR";
asLeakTesterTestEvaluation[25] := "PROG ERROR";
asLeakTesterTestEvaluation[26] := "CALCULATION ERROR";
asLeakTesterTestEvaluation[27] := "INVALID PROGRAM SELECTED";
asLeakTesterTestEvaluation[28] := "INVALID CALIBRATION DATA";
asLeakTesterTestEvaluation[29] := "INVALID I/O CONFIGURATION";
asLeakTesterTestEvaluation[30] := "I/O FAULT";
asLeakTesterTestEvaluation[31] := "CAL REQUIRED - LIMIT EXCEEDED";
asLeakTesterTestEvaluation[32] := "CAL REQUIRED - PARAM CHANGED";
asLeakTesterTestEvaluation[33] := "MIN PERF FACTOR ERROR";
asLeakTesterTestEvaluation[34] := "MASTER+LEAK LOSS<MASTER LOSS";
asLeakTesterTestEvaluation[35] := "MASTER LOSS>MAX M+L LOSS";
asLeakTesterTestEvaluation[36] := "MASTER+LEAK LOSS>MAX M+L LOSS";
asLeakTesterTestEvaluation[37] := "MASTER FLOW>MAX M+L FLOW";
asLeakTesterTestEvaluation[38] := "MASTER FLOW<MIN MASTER FLOW";
asLeakTesterTestEvaluation[39] := "MASTER+LEAK FLOW>MAX M+L FLOW";
asLeakTesterTestEvaluation[40] := "MASTER FLOW>MAX MASTER FLOW";
asLeakTesterTestEvaluation[41] := "MASTER+LEAK FLOW>MAX MASTER FLOW";
asLeakTesterTestEvaluation[42] := "MASTER LOSS<MIN MASTER LOSS";
asLeakTesterTestEvaluation[43] := "MASTER LOSS>MAX MASTER LOSS";
asLeakTesterTestEvaluation[44] := "STOP BUTTON PRESSED";
asLeakTesterTestEvaluation[45] := "STOP INPUT RECEIVED";
asLeakTesterTestEvaluation[46] := "ERROR: STOP INPUT HIGH";
asLeakTesterTestEvaluation[47] := "START COMMON INPUT LOW";
asLeakTesterTestEvaluation[48] := "ERROR: ANTI-TIE DOWN";
asLeakTesterTestEvaluation[49] := "ERROR: PART NOT PRESENT";
asLeakTesterTestEvaluation[50] := "ERROR: PART NOT CHANGED";
asLeakTesterTestEvaluation[51] := "EXT SWITCH DID NOT GO LOW";
asLeakTesterTestEvaluation[52] := "EXT SWITCH DID NOT GO HIGH";
asLeakTesterTestEvaluation[53] := "ERROR: TOOLING NOT RESET";
asLeakTesterTestEvaluation[54] := "ERROR: TOOLING NOT EXTENDED";
asLeakTesterTestEvaluation[55] := "ERROR: TOOLING NOT RETRACTED";
asLeakTesterTestEvaluation[56] := "TOOLING RESET";
asLeakTesterTestEvaluation[57] := "ERROR: PART MARK FAULT";
asLeakTesterTestEvaluation[58] := "PART NOT FULL";
asLeakTesterTestEvaluation[59] := "PART NOT EXHAUSTED";
asLeakTesterTestEvaluation[60] := "PART NOT STABILIZED";
asLeakTesterTestEvaluation[61] := "AUTOSETUP SEQ COMPLETE";
asLeakTesterTestEvaluation[62] := "DP TRANSDUCER ZERO BAD";
asLeakTesterTestEvaluation[63] := "DP TRANSDUCER OVER-RANGE";
asLeakTesterTestEvaluation[64] := "ERROR: TWO-INPUT REQ TO START";
asLeakTesterTestEvaluation[65] := "ERROR: BARCODE REQ TO START";
asLeakTesterTestEvaluation[66] := "DP TRANSDUCER FAULT";
asLeakTesterTestEvaluation[67] := "ERROR: NO LINKS DEFINED";
asLeakTesterTestEvaluation[68] := "ERROR: LINK EXECUTION LOOP";
asLeakTesterTestEvaluation[69] := "ERROR: LINK PROG IS PARENT";
asLeakTesterTestEvaluation[70] := "ERROR: LINK PROG UNDEFINED";
asLeakTesterTestEvaluation[71] := "ERROR: DISSIMILAR LINK ORDER";
asLeakTesterTestEvaluation[72] := "ERROR: DUPLICATE TARGET LINK";
asLeakTesterTestEvaluation[73] := "CAL PROGRAM ACCEPT";
asLeakTesterTestEvaluation[74] := "CAL PROGRAM REJECT";
asLeakTesterTestEvaluation[75] := "PRESSURE TRANSDUCER FAULT";
asLeakTesterTestEvaluation[76] := "NO EVENT OCCURRED";
asLeakTesterTestEvaluation[77] := "SYSTEM PRESSURE EXCEEDED";
asLeakTesterTestEvaluation[78] := "PRESSURE SELECT CONFIG ERROR";
asLeakTesterTestEvaluation[79] := "LEAK STD SELECT CONFIG ERROR";
asLeakTesterTestEvaluation[80] := "VENT PART RESET TOOLING";
asLeakTesterTestEvaluation[81] := "TRANSDUCER CAL COMPLETE";
asLeakTesterTestEvaluation[82] := "TRANSDUCER CAL ERROR";
asLeakTesterTestEvaluation[83] := "TRANSDUCER VERIFY COMPLETE";
asLeakTesterTestEvaluation[84] := "ELEC REGULATOR CAL COMPLETE";
asLeakTesterTestEvaluation[85] := "ELEC REGULATOR CAL ERROR";
asLeakTesterTestEvaluation[86] := "SYSTEM ERROR - SERVICE REQ";
asLeakTesterTestEvaluation[87] := "TEST PORT SELECT CONFIG ERROR";
asLeakTesterTestEvaluation[88] := "SOURCE PRESSURE EXCEEDED";
asLeakTesterTestEvaluation[89] := "PRE-PRESSURE LOW";
asLeakTesterTestEvaluation[90] := "PRE-PRESSURE HIGH";
asLeakTesterTestEvaluation[91] := "ERROR: SNIFFER NOT READY";
asLeakTesterTestEvaluation[92] := "SNIFFER UNITS MISMATCH";
asLeakTesterTestEvaluation[93] := "SNIFFER MODE MISMATCH";
asLeakTesterTestEvaluation[94] := "T-GAS BACKGROUND FAULT";
asLeakTesterTestEvaluation[95] := "T-GAS MIN LEAK RATE FAULT";
asLeakTesterTestEvaluation[96] := "T-GAS CHAMBER CLEANUP FAULT";
asLeakTesterTestEvaluation[97] := "SNIFFER TYPE MISMATCH";
asLeakTesterTestEvaluation[98] := "SNIFFER READY INPUT FAULT";
asLeakTesterTestEvaluation[99] := "CHAMBER EVACUATION FAULT";
asLeakTesterTestEvaluation[100] := "CHAMBER RISE FAULT";
asLeakTesterTestEvaluation[101] := "SCALE CONFIG ERROR";
asLeakTesterTestEvaluation[102] := "SCALE NOT READY";
asLeakTesterTestEvaluation[103] := "SCALE NOT STABLE";
asLeakTesterTestEvaluation[104] := "SCALE WEIGHT LOW";
asLeakTesterTestEvaluation[105] := "SCALE WEIGHT HIGH";
asLeakTesterTestEvaluation[106] := "WEIGHT BELOW MIN";
asLeakTesterTestEvaluation[107] := "WEIGHT ABOVE MAX";
asLeakTesterTestEvaluation[108] := "ATMOSPHERIC PRESSURE COMPLETE";
asLeakTesterTestEvaluation[109] := "ATMOSPHERIC PRESSURE ERROR";
asLeakTesterTestEvaluation[110] := "EXTERNAL XDCR PRESS";
asLeakTesterTestEvaluation[111] := "MAN FILL SWITCH";
asLeakTesterTestEvaluation[112] := "ISOLATION FAILURE";
asLeakTesterTestEvaluation[113] := "LD ZERO < MIN";
asLeakTesterTestEvaluation[114] := "LD ZERO > MAX";
asLeakTesterTestEvaluation[115] := "LD LEAK < MIN";
asLeakTesterTestEvaluation[116] := "LD LEAK > MAX";
asLeakTesterTestEvaluation[117] := "PROCESS FAULT";
asLeakTesterTestEvaluation[118] := "POWER RESET";
asLeakTesterTestEvaluation[119] := "INVALID INPUT CONFIGURATION";
asLeakTesterTestEvaluation[120] := "INPUT INITIAL STATE ERROR";
asLeakTesterTestEvaluation[121] := "MASS SPEC CONTAMINATION";
asLeakTesterTestEvaluation[122] := "CHAMBER PRESSURE HIGH";
asLeakTesterTestEvaluation[123] := "CHAMBER CROSSOVER INPUT FAULT";
asLeakTesterTestEvaluation[124] := "CHAMBER RISE INPUT FAULT";
asLeakTesterTestEvaluation[125] := "T-GAS PART FILL FAULT";
asLeakTesterTestEvaluation[126] := "T-GAS LEAK STD FAULT";
asLeakTesterTestEvaluation[127] := "MASTER+LEAK LOSS<MIN M+L LOSS";
asLeakTesterTestEvaluation[128] := "LEAK LOSS<MIN LEAK LOSS";
asLeakTesterTestEvaluation[129] := "LEAK LOSS>MAX LEAK LOSS";
asLeakTesterTestEvaluation[130] := "MASTER+LEAK FLOW<MIN M+L FLOW";
asLeakTesterTestEvaluation[131] := "LEAK FLOW<MIN LEAK FLOW";
asLeakTesterTestEvaluation[132] := "LEAK FLOW > MAX LEAK FLOW";
asLeakTesterTestEvaluation[133] := "MASTER+LEAK PART COMPLETE";
asLeakTesterTestEvaluation[134] := "VALVE LOAD FAULT";
asLeakTesterTestEvaluation[135] := "ERROR: INSTRUMENT NOT ENABLED";
asLeakTesterTestEvaluation[136] := "CHARGE PRESSURE LOW";
asLeakTesterTestEvaluation[137] := "CHARGE PRESSURE HIGH";
END_ACTION

ACTION ACT_LeakTesterUnit:
asLeakTesterUnit[0] := "NO DATA";
asLeakTesterUnit[1] := "atm";
asLeakTesterUnit[2] := "bar";
asLeakTesterUnit[3] := "cmHg";
asLeakTesterUnit[4] := "inHg";
asLeakTesterUnit[5] := "kPa";
asLeakTesterUnit[6] := "MPa";
asLeakTesterUnit[7] := "mbar";
asLeakTesterUnit[8] := "mmHg";
asLeakTesterUnit[9] := "Pa";
asLeakTesterUnit[10] := "Torr";
asLeakTesterUnit[11] := "psig";
asLeakTesterUnit[12] := "psiv";
asLeakTesterUnit[13] := "iWC";
asLeakTesterUnit[14] := "cmWC";
asLeakTesterUnit[15] := "mmWC";
asLeakTesterUnit[16] := "ksc";
asLeakTesterUnit[17] := "psia";
asLeakTesterUnit[18] := "datm";
asLeakTesterUnit[19] := "dbar";
asLeakTesterUnit[20] := "dcmHg";
asLeakTesterUnit[21] := "dinHg";
asLeakTesterUnit[22] := "dkPa";
asLeakTesterUnit[23] := "dMpa";
asLeakTesterUnit[24] := "dmbar";
asLeakTesterUnit[25] := "dmmHg";
asLeakTesterUnit[26] := "dPa";
asLeakTesterUnit[27] := "dTorr";
asLeakTesterUnit[28] := "dpsig";
asLeakTesterUnit[29] := "dpsiv";
asLeakTesterUnit[30] := "diWC";
asLeakTesterUnit[31] := "dcmWC";
asLeakTesterUnit[32] := "dmmWC";
asLeakTesterUnit[33] := "dksc";
asLeakTesterUnit[34] := "dpsi";
asLeakTesterUnit[35] := "sccm";
asLeakTesterUnit[36] := "sces";
asLeakTesterUnit[37] := "scch";
asLeakTesterUnit[38] := "scfm";
asLeakTesterUnit[39] := "slpm";
asLeakTesterUnit[40] := "slps";
asLeakTesterUnit[41] := "scfh";
asLeakTesterUnit[42] := "scfs";
asLeakTesterUnit[43] := "slph";
asLeakTesterUnit[44] := "gs";
asLeakTesterUnit[45] := "gm";
asLeakTesterUnit[46] := "degC";
asLeakTesterUnit[47] := "degF";
asLeakTesterUnit[48] := "degK";
asLeakTesterUnit[49] := "hour";
asLeakTesterUnit[50] := "min";
asLeakTesterUnit[51] := "sec";
asLeakTesterUnit[52] := "msec";
asLeakTesterUnit[53] := "yr";
asLeakTesterUnit[54] := "mth";
asLeakTesterUnit[55] := "wk";
asLeakTesterUnit[56] := "day";
asLeakTesterUnit[57] := "cc";
asLeakTesterUnit[58] := "cin";
asLeakTesterUnit[59] := "l";
asLeakTesterUnit[60] := "gal";
asLeakTesterUnit[61] := "mL";
asLeakTesterUnit[62] := "in";
asLeakTesterUnit[63] := "mic";
asLeakTesterUnit[64] := "cm";
asLeakTesterUnit[65] := "mm";
asLeakTesterUnit[66] := "M";
asLeakTesterUnit[67] := "thou";
asLeakTesterUnit[68] := "mil";
asLeakTesterUnit[69] := "V";
asLeakTesterUnit[70] := "mV";
asLeakTesterUnit[71] := "uV";
asLeakTesterUnit[72] := "A";
asLeakTesterUnit[73] := "mA";
asLeakTesterUnit[74] := "uA";
asLeakTesterUnit[75] := "dB";
asLeakTesterUnit[76] := "bits";
asLeakTesterUnit[77] := "ppm";
asLeakTesterUnit[78] := "PF";
asLeakTesterUnit[79] := "%";
asLeakTesterUnit[80] := "unit";
asLeakTesterUnit[81] := "cnts";
asLeakTesterUnit[82] := "atm/s";
asLeakTesterUnit[83] := "bar/s";
asLeakTesterUnit[84] := "cHg/s";
asLeakTesterUnit[85] := "inHg/s";
asLeakTesterUnit[86] := "kPa/s";
asLeakTesterUnit[87] := "psi/s";
asLeakTesterUnit[88] := "iWC/s";
asLeakTesterUnit[89] := "cWC/s";
asLeakTesterUnit[90] := "mWC/s";
asLeakTesterUnit[91] := "ksc/s";
asLeakTesterUnit[92] := "g/a";
asLeakTesterUnit[93] := "oz/yr";
asLeakTesterUnit[94] := "ppm";
asLeakTesterUnit[95] := "mbl/s";
asLeakTesterUnit[96] := "Pam/s";
asLeakTesterUnit[97] := "acc/s";
asLeakTesterUnit[98] := "Trl/s";
asLeakTesterUnit[99] := "Pam/h";
asLeakTesterUnit[100] := "gr/yr";
asLeakTesterUnit[101] := "lb/yr";
asLeakTesterUnit[102] := "acc/m";
asLeakTesterUnit[103] := "kg";
asLeakTesterUnit[104] := "g";
asLeakTesterUnit[105] := "lb";
asLeakTesterUnit[106] := "oz";
asLeakTesterUnit[107] := "MPa/s";
asLeakTesterUnit[108] := "mb/s";
asLeakTesterUnit[109] := "mHg/s";
asLeakTesterUnit[110] := "pa/s";
asLeakTesterUnit[111] := "MPa/s";
END_ACTION

ACTION ACT_LiveSegmentCode:
asLeakTesterSegments[0] := "NO DATA";
asLeakTesterSegments[1] := "INTERN PreSeq";
asLeakTesterSegments[2] := "Intern PostSeq";
asLeakTesterSegments[3] := "Intern EmptySeq";
asLeakTesterSegments[4] := "Intern - Evaluate Part Result";
asLeakTesterSegments[5] := "Setup - Pre-Seq";
asLeakTesterSegments[6] := "Setup - Post-Seq";
asLeakTesterSegments[7] := "Setup - Pressure Select";
asLeakTesterSegments[8] := "Setup - Manifold Fill";
asLeakTesterSegments[9] := "Setup - Manifold Isolate";
asLeakTesterSegments[10] := "Setup - Manifold Exhaust";
asLeakTesterSegments[11] := "Prefill til Pressure";
asLeakTesterSegments[12] := "Prefill";
asLeakTesterSegments[13] := "Prefill Pre-Pressure";
asLeakTesterSegments[14] := "Prefill - Charge Volume";
asLeakTesterSegments[15] := "Fill References";
asLeakTesterSegments[16] := "Fill (without pressure monitoring)";
asLeakTesterSegments[17] := "Fill Ramp";
asLeakTesterSegments[18] := "Fill Tracer";
asLeakTesterSegments[19] := "Fill Tracer Gross";
asLeakTesterSegments[20] := "Fill Step";
asLeakTesterSegments[21] := "Fill Evac";
asLeakTesterSegments[22] := "Fill Clean";
asLeakTesterSegments[23] := "Fill til Full";
asLeakTesterSegments[24] := "Stabilize Tracer";
asLeakTesterSegments[25] := "Stabilize Tracer Gross";
asLeakTesterSegments[26] := "Stabilize DP Xder Balance";
asLeakTesterSegments[27] := "Stabilize Evac";
asLeakTesterSegments[28] := "Stabilize Step Dwell";
asLeakTesterSegments[29] := "Stabilize Chamber Cleanup";
asLeakTesterSegments[30] := "Stabilize til Slope";
asLeakTesterSegments[31] := "Stabilize DP";
asLeakTesterSegments[32] := "Stabilize Xder Test";
asLeakTesterSegments[33] := "Stabilize Flow";
asLeakTesterSegments[34] := "Stabilize References Volume";
asLeakTesterSegments[35] := "Stabilize Tracer Wait";
asLeakTesterSegments[36] := "Stabilize Balance DP";
asLeakTesterSegments[37] := "Pressure Decay - Leak Standard Test";
asLeakTesterSegments[38] := "Rate Pressure Loss Test";
asLeakTesterSegments[39] := "Occlusion Test (Backpressure)";
asLeakTesterSegments[40] := "Percent References Volume Test";
asLeakTesterSegments[41] := "Pressure Loss Test";
asLeakTesterSegments[42] := "Ramp Pressure Event Test";
asLeakTesterSegments[43] := "Proof Test";
asLeakTesterSegments[44] := "Ramp Flow Event Test";
asLeakTesterSegments[45] := "Refrigerant Fill";
asLeakTesterSegments[46] := "Ramp Digital Input Event Test";
asLeakTesterSegments[47] := "Sniffer Test";
asLeakTesterSegments[48] := "Sniffer Gross Test";
asLeakTesterSegments[49] := "Step Proof";
asLeakTesterSegments[50] := "Differential Pressure Decay - Leak Standard Test";
asLeakTesterSegments[51] := "Evac Test";
asLeakTesterSegments[52] := "Differential Pressure Decay Test";
asLeakTesterSegments[53] := "Differential Pressure Decay Test (no absl pressure)";
asLeakTesterSegments[54] := "Precise Mass Flow Test (Differential Flow)";
asLeakTesterSegments[55] := "Mass Flow Test";
asLeakTesterSegments[56] := "Mass Flow - Leak Rate Test";
asLeakTesterSegments[57] := "Differential Pressure Decay - Leak Standard Test (no absl pressure)";
asLeakTesterSegments[58] := "Differential Pressure Decay - Leak Rate (volume calculated)";
asLeakTesterSegments[59] := "Pressure Switch Test";
asLeakTesterSegments[60] := "Transducer Test";
asLeakTesterSegments[61] := "Pressure Verify";
asLeakTesterSegments[62] := "Exhaust";
asLeakTesterSegments[63] := "Exhaust til Pressure";
asLeakTesterSegments[64] := "Exhaust til Input";
asLeakTesterSegments[65] := "Exhaust til Analog Input";
asLeakTesterSegments[66] := "Exhaust til Slope";
asLeakTesterSegments[67] := "Exhaust til Empty";
asLeakTesterSegments[68] := "Exhaust - Re-Evacuate";
asLeakTesterSegments[69] := "Exhaust - T-Gas";
asLeakTesterSegments[70] := "Exhaust - Chamber Output Rest";
asLeakTesterSegments[71] := "Verify Pressure";
asLeakTesterSegments[72] := "Verify Pressure after Delay";
asLeakTesterSegments[73] := "Verify Input";
asLeakTesterSegments[74] := "Verify Input after Delay";
asLeakTesterSegments[75] := "Verify Analog Input";
asLeakTesterSegments[76] := "Verify Analog Input after Delay";
asLeakTesterSegments[77] := "Verify Slope";
asLeakTesterSegments[78] := "Verify Slope after Delay";
asLeakTesterSegments[79] := "Drive Output";
asLeakTesterSegments[80] := "Drive Output Period";
asLeakTesterSegments[81] := "Drive Analog Output";
asLeakTesterSegments[82] := "Drive Analog Output Period";
asLeakTesterSegments[83] := "Drive Valve";
asLeakTesterSegments[84] := "Drive Valve Period";
asLeakTesterSegments[85] := "Link Control";
asLeakTesterSegments[86] := "Link Decision";
asLeakTesterSegments[87] := "Autorun Relax";
asLeakTesterSegments[88] := "Calibration Relax";
asLeakTesterSegments[89] := "Delay";
asLeakTesterSegments[90] := "Pressure Transducer Zero";
asLeakTesterSegments[91] := "Flow Transducer Zero";
asLeakTesterSegments[92] := "Differential Pressure Transducer Zero";
asLeakTesterSegments[93] := "Pressure Select (Range Only)";
asLeakTesterSegments[94] := "Pressure Select (Evac)";
asLeakTesterSegments[95] := "Pressure Select";
asLeakTesterSegments[96] := "Pressure Select (Ramp)";
asLeakTesterSegments[97] := "Pressure Select (Tracer)";
asLeakTesterSegments[98] := "Pressure Select (Clean)";
asLeakTesterSegments[99] := "Pressure Select (None)";
asLeakTesterSegments[100] := "Tooling Motion Control";
asLeakTesterSegments[101] := "Tooling Motion Extend";
asLeakTesterSegments[102] := "Tooling Motion Retract";
asLeakTesterSegments[103] := "Tooling Part Mark";
asLeakTesterSegments[104] := "Tooling Seal Extend";
asLeakTesterSegments[105] := "Tooling Seal Retract";
asLeakTesterSegments[106] := "External Volume";
asLeakTesterSegments[107] := "Setup - Set Regulator";
asLeakTesterSegments[108] := "Setup - Electronic Regulator Analyze";
asLeakTesterSegments[109] := "Setup - Electronic Regulator Zero";
asLeakTesterSegments[110] := "Setup - Electronic Regulator Setpoint";
asLeakTesterSegments[111] := "Setup - Transducer Residual";
asLeakTesterSegments[112] := "Setup - Pressure Transducer Zero";
asLeakTesterSegments[113] := "Setup - Flow Transducer Zero";
asLeakTesterSegments[114] := "Setup - Pressure Transducer Setpoint";
asLeakTesterSegments[115] := "Setup - Flow Transducer Setpoint";
asLeakTesterSegments[116] := "Setup - DP Transducer Setpoint";
asLeakTesterSegments[117] := "Setup - Pressure Transducer Verification";
asLeakTesterSegments[118] := "Setup - Flow Transducer Verification";
asLeakTesterSegments[119] := "Setup - Sniffer Init 1";
asLeakTesterSegments[120] := "Setup - Sniffer Init 2";
asLeakTesterSegments[121] := "Setup - Sniffer Idle";
asLeakTesterSegments[122] := "Setup - Mix Verification";
asLeakTesterSegments[123] := "Setup - Scale Init";
asLeakTesterSegments[124] := "Setup - Atmospheric Pressure Check";
asLeakTesterSegments[125] := "Setup - DP Transducer Zero";
asLeakTesterSegments[126] := "Setup - DP Transducer Verification";
asLeakTesterSegments[127] := "Begin Chamber Functions";
asLeakTesterSegments[128] := "Chamber - hardvac control";
asLeakTesterSegments[129] := "Chamber - blower control";
asLeakTesterSegments[130] := "Chamber - inlet blower on";
asLeakTesterSegments[131] := "Chamber - inlet blower off";
asLeakTesterSegments[132] := "Chamber - circulation on";
asLeakTesterSegments[133] := "Chamber - outlet blower on";
asLeakTesterSegments[134] := "Chamber - outlet blower off";
asLeakTesterSegments[135] := "Chamber - circulation off";
asLeakTesterSegments[136] := "Chamber - accumulation rest";
asLeakTesterSegments[137] := "Chamber - clamshell purge rings control";
asLeakTesterSegments[138] := "Chamber - clamshell purge rings option";
asLeakTesterSegments[139] := "Chamber - clamshell purge rings rest";
asLeakTesterSegments[140] := "Chamber - Exh";
asLeakTesterSegments[141] := "Chamber - vent off";
asLeakTesterSegments[142] := "Chamber - evacuate on";
asLeakTesterSegments[143] := "Chamber - evacuate off";
asLeakTesterSegments[144] := "Chamber - pre-purge";
asLeakTesterSegments[145] := "Refrigerant CS Isolation";
asLeakTesterSegments[146] := "Refrigerant Stabilize";
asLeakTesterSegments[147] := "Refrigerant Part Switch";
asLeakTesterSegments[148] := "Refrigerant Vent";
asLeakTesterSegments[149] := "Refrigerant Iso Off";
asLeakTesterSegments[150] := "Stabilize Scale";
asLeakTesterSegments[151] := "Refrigerant Manual Fill";
asLeakTesterSegments[152] := "Refrigerant Evac";
END_ACTION

ACTION ACT_Precision:
asLeakTesterPrecision[0] := "NO DATA";
asLeakTesterPrecision[1] := "Digits of precision: X";
asLeakTesterPrecision[2] := "Digits of precision: X.X";
asLeakTesterPrecision[3] := "Digits of precision: X.XX";
asLeakTesterPrecision[4] := "Digits of precision: X.XXX";
asLeakTesterPrecision[5] := "Digits of precision: X.XXXX";
asLeakTesterPrecision[6] := "Digits of precision: X.XXXXX";
END_ACTION

ACTION ACT_ProgramEvaluation:
asLeakTesterProgramEvaluation[0] := "NO DATA";
asLeakTesterProgramEvaluation[1] := "TEST PASSED";
asLeakTesterProgramEvaluation[2] := "TEST FAILED";
asLeakTesterProgramEvaluation[3] := "TEST ERROR";
asLeakTesterProgramEvaluation[4] := "TEST SKIPPED";
asLeakTesterProgramEvaluation[5] := "TEST FAILED - LEVEL 1";
asLeakTesterProgramEvaluation[6] := "TEST FAILED - LEVEL 2";
asLeakTesterProgramEvaluation[7] := "TEST FAILED - LEVEL 3";
asLeakTesterProgramEvaluation[8] := "AUTO-CAL MASTER PART";
asLeakTesterProgramEvaluation[9] := "AUTO-CAL LEAK STANDARD PART";
asLeakTesterProgramEvaluation[10] := "TEST FAILED - NO EVENT";
asLeakTesterProgramEvaluation[11] := "TEST COMPLETE";
END_ACTION

ACTION ACT_TestType:
asLeakTesterTestType[0] := "NO DATA";
asLeakTesterTestType[1] := "Pressure Decay - Leak Standard Test";
asLeakTesterTestType[2] := "Rate of Pressure Loss Test";
asLeakTesterTestType[3] := "Occlusion Test (Backpressure)";
asLeakTesterTestType[4] := "Percent of Reference Volume Tes";
asLeakTesterTestType[5] := "Pressure Loss Test";
asLeakTesterTestType[6] := "Ramp to Pressure Event Test";
asLeakTesterTestType[7] := "Proof Test";
asLeakTesterTestType[8] := "Ramp to Flow Event Test";
asLeakTesterTestType[9] := "Refrigerant Fill";
asLeakTesterTestType[10] := "Ramp to Digital Input Event Test";
asLeakTesterTestType[11] := "Sniffer Test";
asLeakTesterTestType[12] := "";
asLeakTesterTestType[13] := "Sniffer Gross Test";
asLeakTesterTestType[14] := "Step Proof";
asLeakTesterTestType[15] := "Differential Pressure Decay - Leak | Standard Test";
asLeakTesterTestType[16] := "Evac Test";
asLeakTesterTestType[17] := "Differential Pressure Decay Test";
asLeakTesterTestType[18] := "Differential Pressure Decay Test (no abs pressure)";
asLeakTesterTestType[19] := "Precise Mass Flow Test (Differential Flow)";
asLeakTesterTestType[20] := "Mass Flow Test";
asLeakTesterTestType[21] := "Mass Flow - Leak Rate Test";
asLeakTesterTestType[22] := "Differential Pressure Decay - Leak Standard Test (no abs pressure)";
asLeakTesterTestType[23] := "Differential Pressure Decay - Leak Rate (volume calculated)";
asLeakTesterTestType[24] := "Pressure Switch Test";
asLeakTesterTestType[25] := "Transducer Test";
END_ACTION

END_PROGRAM

// ---- POUs/B_HightTest/PRG_HeightTest.TcPOU
PROGRAM PRG_HeightTest
VAR
	//FUNCTION
	fbHeightMeasurement2						: FB_HeightMeasurement2;
	
	
	bEnable										: BOOL;
	bEnableo									: BOOL;
	bMeasurementRequest							: BOOL;
	bSet										: BOOL;
	bAcknowledge								: BOOL;
	bManualMode									: BOOL;
	bBusy										: BOOL;
	bComplete									: BOOL;

//TrigTim

	rtrigCaseTriger			: ARRAY[1..20] OF R_TRIG;
	tonCaseDelay			: ARRAY[1..10] OF TON;

	
	
END_VAR


VAR_IN_OUT
	stStationStruct          	: ST_StandardStationStruct;
	
END_VAR
VAR PERSISTENT
stHeightMeasurement2						: ST_HeightMeasurement2;
END_VAR

ACT_IOLink();
ACT_TimTrig();
ACT_Statistics();
ACT_ProbesPosition();

(************** Station in Home Position **************************)
stStationStruct.bStationHomed :=  (stStationStruct.nState = 1000);

(******************************************************************)
stStationStruct.bStationComplete := stStationStruct.nState = 1220;
stStationStruct.bStationHomingRequest := stStationStruct.nState = 200;
stStationStruct.bStationWaitOnRequest := stStationStruct.nState = 1000; 
stStationStruct.bStationInitDone := stStationStruct.nState = 400;
stStationStruct.bStationInProgressInit := stStationStruct.nState >= 200 AND stStationStruct.nState <= 900;
stStationStruct.bStationInProgress :=  stStationStruct.nState > 1000 AND stStationStruct.nState < 1900;
stStationStruct.bStationWaitOnInit := stStationStruct.nState = 100; 
//stStationStruct.bStationAcknowledge := stStationStruct.nState = 200 OR stStationStruct.nState = 1100;
stStationStruct.bStationNotMoving := stStationStruct.nState = 100 OR stStationStruct.nState = 1000 OR stStationStruct.nState = 1240;
(******************************************************************)
(***************** Counter *************)


(***************************************)

IF rtrigCaseTriger[5].Q THEN
	stStationStruct.nState := 100;
END_IF

(***************************************)


CASE stStationStruct.nState OF
100:
bMeasurementRequest := FALSE;
IF stStationStruct.bStationInitRequest THEN
	stStationStruct.nState:= 300;
END_IF

300:
IF tonCaseDelay[1].Q THEN
   stStationStruct.nState:= 400;	
END_IF
400:
	stStationStruct.nState:= 1000;

//============== Homed ========================================================

1000:

IF GVL_HMI_GLOBAL.bResetPassAndFail THEN
	bEnable 			:= FALSE;
	bAcknowledge 		:= FALSE;
	bMeasurementRequest	:= FALSE;
	GVL_MASTER.stNest.bHeightPass := FALSE;
	GVL_MASTER.stNest.sHeightHMI := "";
	GVL_MASTER.stNest.bHeightReject := FALSE;

END_IF
IF stStationStruct.bStationRequest AND stStationStruct.bNoCycleStopRequest THEN
   	stStationStruct.nState := 1010;  
ELSIF (stStationStruct.bStationManualRequestHMI OR GVL_MASTER.bManualModeTrigger) AND stStationStruct.bNoCycleStopRequest THEN
   stStationStruct.nState := 4000; // Manual Mode
ELSIF stStationStruct.bStationAbort THEN
	   stStationStruct.nState := 100;	   
END_IF
1010:
bEnable := TRUE;
IF tonCaseDelay[2].Q THEN
	stStationStruct.nState:= 1100;
END_IF
1100:
IF bEnableo THEN
	stStationStruct.nState:= 1110;
END_IF
1110:
bMeasurementRequest := TRUE;
IF NOT bBusy AND bComplete THEN
	bMeasurementRequest := FALSE;
	bAcknowledge		:= TRUE;
	stStationStruct.nState:= 1120;
END_IF
1120: // JOB PASS / JOB FAIL
bAcknowledge			:= FALSE;

IF bComplete AND NOT bBusy  THEN
	GVL_MASTER.stNest.bHeightPass := GVL_HMI_GLOBAL.aGeneralPassHeightTest[5];
	GVL_MASTER.stNest.bHeightReject := GVL_HMI_GLOBAL.aGeneralFailHeightTest[5];
	
	IF GVL_MASTER.stNest.bHeightPass THEN
		GVL_MASTER.stNest.sHeightHMI 	:= "Pass";
		GVL_MASTER.stNest.bHeightPass := TRUE;
		GVL_MASTER.stNest.bHeightReject := FALSE;
	ELSIF  GVL_MASTER.stNest.bHeightReject THEN
		
		GVL_MASTER.stNest.sHeightHMI 	:= "Fail";
		GVL_MASTER.stNest.bHeightPass := FALSE;
		GVL_MASTER.stNest.bHeightReject := TRUE;
	END_IF
	
	stStationStruct.nState:= 1220;
END_IF
1220:

IF tonCaseDelay[5].Q THEN
	stStationStruct.nState:= 1240;
END_IF

1240:
IF (tonCaseDelay[3].Q AND NOT stStationStruct.bStationManualRequestHMI OR GVL_MASTER.bHeightTestacknowledge) OR NOT stStationStruct.bNoCycleStopRequest THEN
	stStationStruct.nState:= 1000;
ELSIF tonCaseDelay[3].Q AND stStationStruct.bStationManualRequestHMI AND stStationStruct.bNoCycleStopRequest THEN
	stStationStruct.nState:= 4000;
END_IF


4000:
IF NOT stStationStruct.bStationManualRequestHMI AND NOT GVL_MASTER.bManualModeTrigger THEN
	stStationStruct.nState := 1000;
	bEnable				:= FALSE;
	bManualMode			:= FALSE;
ELSIF stStationStruct.bStationAbort THEN
	 stStationStruct.nState := 100;
	 bEnable				:= FALSE;
	bManualMode			:= FALSE;
ELSE 
bManualMode			:= TRUE;
bEnable				:= TRUE;	
END_IF



END_CASE

ACTION ACT_IOLink:

stHeightMeasurement2.aSensorCurrentValue[1]		:= DINT_TO_REAL(GVL_IO.dw_B08_DL_PN1.gt2_1_1CurrentValue);
stHeightMeasurement2.aSensorCurrentValue[2]		:= DINT_TO_REAL(GVL_IO.dw_B08_DL_PN1.gt2_1_2CurrentValue);
stHeightMeasurement2.aSensorCurrentValue[3]		:= DINT_TO_REAL(GVL_IO.dw_B08_DL_PN1.gt2_1_3CurrentValue);
stHeightMeasurement2.aSensorCurrentValue[4]		:= DINT_TO_REAL(GVL_IO.dw_B08_DL_PN1.gt2_2CurrentValue);

fbHeightMeasurement2(
	
	aSensorCurrentValue							:= stHeightMeasurement2.aSensorCurrentValue,	
	bEnable										:= bEnable,
	bMeasurementRequest							:= bMeasurementRequest,
	bSetFixedPoints								:= GVL_HMI_GLOBAL.bSetSetPointsHeightTest,
	aTolerance									:= stHeightMeasurement2.aTolerance,
	bAcknowledge								:= bAcknowledge,
	nDistanceBetweenPoints						:= stHeightMeasurement2.nDistanceBetweenPoints,
	anDistanceSetPoint							:= stHeightMeasurement2.anDistanceSetPoint,
	bManualMode									:= bManualMode,
	
